							// Ask operator to fill calbox
							GVL_HMI.bCalBoxNeedsAttention := TRUE;
							bCalBoxAttention := TRUE;
	
							// Stop requesting until operator continues
							bRequestWeight := FALSE;
	
							eStepResume := E_CalibStep.CHECKING_WEIGH;
							eStep       := E_CalibStep.CALBOX_ATTENTION;
	
						ELSE
							// Proceed
							bBoxWeightOK := FALSE;
							bRequestWeight := FALSE;
	
							eStep := E_CalibStep.FEED_HMI_RESULTS;
							rAcceptanceCrit := GVL_Settings.stCalibParameters.rAcceptanceCriteria;
						END_IF
					END_IF
	
					// ------------------------------------------------
					// 4) Always reset the device session AFTER processing
					//    (so bWeightReady doesn't stay stuck TRUE / repeat)
					// ------------------------------------------------
					// If Reset() returns BOOL and you need to ensure completion, you can loop it outside.
					// For now, keep your pattern:
					GVL_Calibration.fbScaleDevice.Reset();
				END_IF
			END_IF
		END_IF
	
	E_CalibStep.FEED_HMI_RESULTS:
	
		FOR i := 1 TO 10 DO
			IF aPumpSettings[i].bSelected THEN
				GVL_HMI.aCalPumpResults[i].eStatus := E_CalibrationStatus.PENDING;
			END_IF
		END_FOR
		
		eStep := E_CalibStep.POSITION_MOTORS;
		
		
	E_CalibStep.POSITION_MOTORS:
	
		sStatus := 'Positioning motors M2 and M3';
		
		// Positioning motors M2 and M3 to calibration position 
		IF NOT bMoveMotorM3 THEN
			bMoveMotorM3 := GVL_Motion.aMotors[3].MoveAbsolute(GVL_Settings.stMachineParam.aM3Position[4], GVL_Settings.stMachineParam.rM3Velocity, GVL_Settings.stMachineParam.rM3Accleration, GVL_Settings.stMachineParam.rM3Deceleration);
		END_IF
		IF NOT bMoveMotorM2 AND bMoveMotorM3 THEN
			bMoveMotorM2 := GVL_Motion.aMotors[2].MoveAbsolute(GVL_Settings.stMachineParam.aM2Position[5], GVL_Settings.stMachineParam.rM2Velocity, GVL_Settings.stMachineParam.rM2Accleration, GVL_Settings.stMachineParam.rM2Deceleration);
		END_IF
	
		IF bMoveMotorM2 AND bMoveMotorM3 THEN
			tonMotorsDelay(in := TRUE, pt := T#200MS);
		END_IF
		
		IF tonMotorsDelay.Q THEN
			tonStepTimeout(IN := FALSE);
			eStep := E_CalibStep.POSITION_VALVES;
		END_IF

    E_CalibStep.POSITION_VALVES:
		//Reset Motors Flags
		bMoveMotorM2 := FALSE;
		bMoveMotorM3 := FALSE;	
		tonMotorsDelay(in := FALSE);
	
		tonStepTimeout(IN := TRUE, PT := tStepTimeout);
        sStatus := 'Positioning valves to Position 6';
		// Positioning the valves to the needles, position 6 
        FOR i := 1 TO 5 DO
            IF NOT bMoveValve[i] THEN
                bMoveValve[i] := GVL_Motion.aValvesObj[i].MoveValve(iPosition := 6, rVelocity := GVL_Motion.aValves[i].rTargetVel, rAcc := GVL_Motion.aValves[i].rAcceleration, rDec := GVL_Motion.aValves[i].rDeceleration);
            END_IF
        END_FOR
       IF bMoveValve[1] AND bMoveValve[2] AND bMoveValve[3] AND bMoveValve[4] AND bMoveValve[5] THEN
			FOR i := 1 TO 5 DO bMoveValve[i] := FALSE; END_FOR
			tonStepTimeout(IN := FALSE);
			eStep := E_CalibStep.FILLJAR_FORWARD; 
		ELSIF tonStepTimeout.Q THEN
			sStatus := 'Timeout while positioning valves';
			eStep := E_CalibStep.ERROR;
		END_IF

	E_CalibStep.FILLJAR_FORWARD:
		
		
		sStatus := CONCAT('Filling up the jar: ', F_JarName(iPumpIndex := iPumpIndex));
		
		IF aPumpSettings[iPumpIndex].bSelected THEN
			IF iPumpIndex = 1 THEN
				rFillJarTotalVol := aPumpSettings[iPumpIndex].rTargetVolume + GVL_Settings.stPumpParameters.iFillolventTubesFactor;
			ELSE
				rFillJarTotalVol := GVL_Settings.stPumpParameters.iFillolventTubesFactor;
			END_IF
			
			GVL_HMI.aCalPumpResults[iPumpIndex].eStatus := E_CalibrationStatus.RUNNING;
			
			//Move Motor M2 for IntoResBottom
			IF NOT bMoveMotorM2 THEN
				bMoveMotorM2 := GVL_Motion.aMotors[2].MoveAbsolute(GVL_Settings.stMachineParam.aM2Position[4], GVL_Settings.stMachineParam.rM2Velocity, GVL_Settings.stMachineParam.rM2Accleration, GVL_Settings.stMachineParam.rM2Deceleration);
			END_IF
				
			rDistanceByVol := F_VolumeToSteps_Path(rVolume := rFillJarTotalVol, iPumpIndex := iPumpIndex, ePath := E_PumpPath.FromCalBox);
			// Filling up the jar to start the calibration
			IF bMoveMotorM2 AND NOT bMovePump THEN
				bMovePump := GVL_Motion.aPumpsRotary[iPumpIndex].MoveRelative(	Distance := rDistanceByVol, 
																				Velocity := GVL_Settings.stPumpParameters.iMeterVelocity * 6, 	//RPM to Degree/sec
																				Acc := GVL_Settings.stPumpParameters.iMeterVelocity * 6,   		//RPM to Degree/sec
																				Dec := GVL_Settings.stPumpParameters.iMeterVelocity * 6			//RPM to Degree/sec
																			 );
			END_IF
	
			IF bMovePump THEN
				tonWeigthStabilization(IN := TRUE, PT := tWeightStable);
				sStatus := 'Waiting for weight stabilization...';
				IF tonWeigthStabilization.Q THEN
					bMovePump := FALSE;
					bMoveMotorM2 := FALSE;
					tonWeigthStabilization(IN := FALSE);
					bRequestWeight := TRUE;
					bWeightReady := FALSE;
					eStep := E_CalibStep.WEIGH_BEFORE;
				END_IF
			END_IF
		ELSE
			// If the pumps was not selected go to next one
			eStep := E_CalibStep.NEXT_PUMP;
		END_IF

	
    E_CalibStep.WEIGH_BEFORE:
		
        sStatus := CONCAT('Pump ', CONCAT(TO_STRING(iPumpIndex), CONCAT(' | Check ', CONCAT(TO_STRING(iReplicate + 1), ' | Taring Scale..'))));
		
		//Move Motor M2 for IntoResWEight
		IF NOT bMoveMotorM2 THEN
			bMoveMotorM2 := GVL_Motion.aMotors[2].MoveAbsolute(GVL_Settings.stMachineParam.aM2Position[6], GVL_Settings.stMachineParam.rM2Velocity, GVL_Settings.stMachineParam.rM2Accleration, GVL_Settings.stMachineParam.rM2Deceleration);
		END_IF
		
        IF bMoveMotorM2 AND bRequestWeight AND NOT bWeightReady THEN
            rScaleWeight := GVL_Calibration.fbScaleDevice.RequestWeight();
            IF GVL_Calibration.fbScaleDevice.bWeightReady THEN
                IF rScaleWeight = 9999.0 THEN
					tonCalDelay(IN := FALSE);
					tonStepTimeout(IN := FALSE);
					tonWeigthStabilization(IN := FALSE);
	
					GVL_HMI.bScaleNeedsAtention := TRUE;
					bScaleAttention := TRUE;
	
					bRequestWeight := FALSE;
					bWeightReady   := FALSE;
	
					eStepResume := E_CalibStep.WEIGH_BEFORE;
					eStep := E_CalibStep.SCALE_ATTENTION;
				ELSE
					rWeightBefore := rScaleWeight;
					
					GVL_calibration.stPumpCalibrationData[GVL_Calibration.iResultIndex].rTareWeigth := rWeightBefore;
					GVL_Calibration.stPumpCalibrationData[GVL_Calibration.iResultIndex].iPumpNumber := TO_USINT(iPumpIndex);
	
					bWeightReady   := TRUE;
					bRequestWeight := NOT GVL_Calibration.fbScaleDevice.Reset();
				END_IF
            END_IF
		END_IF
		IF bWeightReady THEN
			IF (rWeightBefore >= 0 AND rWeightBefore <= 1300) THEN
				GVL_calibration.stPumpCalibrationData[GVL_Calibration.iResultIndex].rTareWeigth := rWeightBefore;
				GVL_Calibration.stPumpCalibrationData[GVL_Calibration.iResultIndex].iPumpNumber := TO_USINT(iPumpIndex);
				rDistanceByVol := 0.0;
				bWeightReady := FALSE;
				bMoveMotorM2 := FALSE;
				eStep := E_CalibStep.WITHDRAW_BACKWARDS;
			ELSE
				eStep := E_CalibStep.ERROR;
			END_IF
		END_IF        

	
    E_CalibStep.WITHDRAW_BACKWARDS:

		sStatus := CONCAT(CONCAT('Pump ',CONCAT(TO_STRING(iPumpIndex),CONCAT(' | Check ',TO_STRING(iReplicate + 1)))),CONCAT(' | Pumping to calibration box: ',CONCAT(TO_STRING(aVolumeSetpoint[iPumpIndex]),' ml')));
		
		//Move Motor M2 for IntoResDispense
		IF NOT bMoveMotorM2 THEN
			bMoveMotorM2 := GVL_Motion.aMotors[2].MoveAbsolute(GVL_Settings.stMachineParam.aM2Position[5], GVL_Settings.stMachineParam.rM2Velocity, GVL_Settings.stMachineParam.rM2Accleration, GVL_Settings.stMachineParam.rM2Deceleration);
		END_IF
		
		aVolumeSetpoint[iPumpIndex] := aPumpSettings[iPumpIndex].rTargetVolume;

		GVL_calibration.stPumpCalibrationData[GVL_Calibration.iResultIndex].rTargetVolume := aPumpSettings[iPumpIndex].rTargetVolume;
		
		rDistanceByVol := F_VolumeToSteps_Path(rVolume := aVolumeSetpoint[iPumpIndex], iPumpIndex := iPumpIndex, ePath := E_PumpPath.FillCalBox );
		
		GVL_calibration.stPumpCalibrationData[GVL_Calibration.iResultIndex].iPumpRevs := TO_UINT(rDistanceByVol/360);
		GVL_HMI.aCalPumpResults[iPumpIndex].iRevsDone := GVL_calibration.stPumpCalibrationData[GVL_Calibration.iResultIndex].iPumpRevs; // Mirror pump revs done to the results table on HMI
		
		IF bMoveMotorM2 AND NOT bMovePump THEN
			bMovePump := GVL_Motion.aPumpsRotary[iPumpIndex].MoveRelative( 	Distance := - rDistanceByVol, 
																			Velocity := GVL_Settings.stPumpParameters.iMeterVelocity * 6, 	//RPM to Degree/sec
																			Acc := GVL_Settings.stPumpParameters.iMeterVelocity * 6, 		//RPM to Degree/sec
																			Dec := GVL_Settings.stPumpParameters.iMeterVelocity				//RPM to Degree/sec
																		 	);
		END_IF
		
		IF bMovePump THEN
			tonWeigthStabilization(in := TRUE, pt := tWeightStable);
			sStatus :='Waiting for weight stabilization...';
			IF bMoveMotorM2 AND tonWeigthStabilization.Q THEN
				bRequestWeight := TRUE;
				bMovePump := FALSE;
				bMoveMotorM2 := FALSE;
				tonWeigthStabilization(IN := FALSE);
				fbLocalSystemTime(bEnable := FALSE);
				bDTReady := FALSE;
				eStep := E_CalibStep.WEIGH_AFTER;
			END_IF
		END_IF


	
    E_CalibStep.WEIGH_AFTER:

		sStatus := CONCAT('Pump ', CONCAT(TO_STRING(iPumpIndex), CONCAT(' | Check ', CONCAT(TO_STRING(iReplicate + 1), ' | Requesting Gross Weight...'))));
	
		//Move Motor M2 for IntoResWeight
		IF NOT bMoveMotorM2 THEN
			bMoveMotorM2 := GVL_Motion.aMotors[2].MoveAbsolute(GVL_Settings.stMachineParam.aM2Position[6], GVL_Settings.stMachineParam.rM2Velocity, GVL_Settings.stMachineParam.rM2Accleration, GVL_Settings.stMachineParam.RM2Deceleration);
		END_IF
		
        IF bMoveMotorM2 AND bRequestWeight AND NOT bWeightReady THEN
            rScaleWeight := GVL_Calibration.fbScaleDevice.RequestWeight();
            IF GVL_Calibration.fbScaleDevice.bWeightReady THEN
                IF rScaleWeight = 9999.0 THEN
					tonCalDelay(IN := FALSE);
					tonStepTimeout(IN := FALSE);
					tonWeigthStabilization(IN := FALSE);
	
					GVL_HMI.bScaleNeedsAtention := TRUE;
					bScaleAttention := TRUE;
	
					bRequestWeight := FALSE;
					bWeightReady   := FALSE;
	
					eStepResume := E_CalibStep.WEIGH_AFTER;
					eStep := E_CalibStep.SCALE_ATTENTION;
				ELSE
					rWeightAfter := rScaleWeight;
					bWeightReady := TRUE;
					// NET (weight delta)
					rWeightDelta := rWeightAfter - rWeightBefore;
	
					// Mirror to logs
					GVL_calibration.stPumpCalibrationData[GVL_Calibration.iResultIndex].rGrossWeigth := rWeightAfter;
					GVL_calibration.stPumpCalibrationData[GVL_Calibration.iResultIndex].rNetWeigth := rWeightDelta;
	
					// Density-based volume
					GVL_calibration.stPumpCalibrationData[GVL_Calibration.iResultIndex].rNetVolume := rWeightDelta / rSolventDensity;
					
					rVolume := GVL_calibration.stPumpCalibrationData[GVL_Calibration.iResultIndex].rNetVolume;
					
					//Getting Sum Values to calculate the average on the end of replicates
					rPumpVolumeSum  := rPumpVolumeSum + rVolume;
					rTareWeightSum  := rTareWeightSum + rWeightBefore;
					rGrossWeightSum := rGrossWeightSum + rWeightAfter;
	
					bRequestWeight := NOT GVL_Calibration.fbScaleDevice.Reset();
				END_IF
			END_IF	
		END_IF	
		
		 // Produce a timestamp: DD-MMM-YYYY HH:MM:SS
        fbLocalSystemTime(bEnable := TRUE, dwCycle := 5);
		
        IF fbLocalSystemTime.bValid THEN
            stLocal := fbLocalSystemTime.systemTime;

            sMMo := F_MonthString(stLocal.wMonth);
            sDD  := F_TwoDigits(stLocal.wDay);
            sHH  := F_TwoDigits(stLocal.wHour);
            sMM  := F_TwoDigits(stLocal.wMinute);
            sSS  := F_TwoDigits(stLocal.wSecond);

			sStamp := CONCAT(sDD, '-');			//DD-
			sStamp := CONCAT(sStamp, sMMo);		//DD-MMM
			sStamp := CONCAT(sStamp, '-');		//DD-MMM-
			sStamp := CONCAT(sStamp, INT_TO_STRING(stLocal.wYear)); //DD-MMM-YYYY
			sStamp := CONCAT(sStamp, ' '); 		//DD-MMM-YYYY 
			sStamp := CONCAT(sStamp, sHH);		//DD-MMM-YYYY HH
			sStamp := CONCAT(sStamp, ':');		//DD-MMM-YYYY HH:
			sStamp := CONCAT(sStamp, sMM);		//DD-MMM-YYYY HH:MM
			sStamp := CONCAT(sStamp, ':');		//DD-MMM-YYYY HH:MM:
			sStamp := CONCAT(sStamp, sSS); 		//DD-MMM-YYYY HH:MM:SS

			bDTReady := TRUE;			
        ELSE
            sStamp := '00000000_000000'; // Fallback if system time is not valid
        END_IF
		
		IF bWeightReady AND bDTReady THEN
			
			rPercentDifference := ((rVolume - aPumpSettings[iPumpIndex].rTargetVolume)  / aPumpSettings[iPumpIndex].rTargetVolume) * 100;
			GVL_Calibration.stPumpCalibrationData[GVL_Calibration.iResultIndex].rDifferenceUl := rVolume - aPumpSettings[iPumpIndex].rTargetVolume;
			GVL_Calibration.stPumpCalibrationData[GVL_Calibration.iResultIndex].dDateTime := sStamp;
			GVL_Calibration.stPumpCalibrationData[GVL_Calibration.iResultIndex].rDifferencePercent := rPercentDifference;
			GVL_Calibration.stPumpCalibrationData[GVL_Calibration.iResultIndex].rCriteria := rAcceptanceCrit;
			
			//pupulate gross weight and net weight
			IF ABS(rPercentDifference) <= rAcceptanceCrit THEN
				aPumpResults[iPumpIndex].eStatus := E_CalibrationStatus.PASSED;
			ELSE
				// Adjust Needed flag 
				bPumpAdjustNeed := TRUE;
			END_IF
			
			iReplicate := iReplicate + 1;
			
			GVL_Calibration.stPumpCalibrationData[GVL_Calibration.iResultIndex].sStep := CONCAT('Check ', TO_STRING(iReplicate));
			
			//DB_Query.state:= E_DB_QUERY_STATE.INSERT_CALIBRATION_VALUES; //Insert new register of data on DB.
			GVL_Calibration.iResultIndex := GVL_Calibration.iResultIndex + 1;
			
			IF iReplicate >= GVL_Settings.stCalibParameters.iReplicatesSetpoint THEN
				
				// Calculating the average pump results
				rPumpAverageVolume  := rPumpVolumeSum / iReplicate;
				rPumpAvgTareWeigth  := rTareWeightSum / iReplicate;
				rPumpAvgGrossWeigth := rGrossWeightSum / iReplicate;
				
				// Mirror the pump status to HMI
				GVL_HMI.aCalPumpResults[iPumpIndex].rAvgNetVolume := rPumpAverageVolume;
				GVL_HMI.aCalPumpResults[iPumpIndex].rAvgTareWeight := rPumpAvgTareWeigth;
				GVL_HMI.aCalPumpResults[iPumpIndex].rAvgGrossWeight := rPumpAvgGrossWeigth;
				
				IF bPumpAdjustNeed THEN
					
					IF GVL_Calibration.iAllowableFailures > iNumberOfAdjusts THEN
						iReplicate := 0;
						iNumberOfAdjusts := iNumberOfAdjusts + 1;
						bPumpAdjustNeed := FALSE;
						DB_Query.state:= E_DB_QUERY_STATE.INSERT_CALIBRATION_VALUES; //Insert new register of data on DB.
						eStep := E_CalibStep.PUMPFACTOR_ADJUST;
					ELSE
						bPumpAdjustNeed := FALSE;
						eStep := E_CalibStep.PUMPFACTOR_FAILED;
					END_IF
					
				ELSE
					GVL_HMI.aCalPumpResults[iPumpIndex].eStatus := E_CalibrationStatus.PASSED;
					eStep := E_CalibStep.EMPTYJAR_BACKWARDS;
				END_IF
			ELSE
				eStep := E_CalibStep.RETURN_FORWARD;
			END_IF
			bMoveMotorM2 := FALSE;
			bWeightReady := FALSE;
		END_IF
		
	E_CalibStep.PUMPFACTOR_ADJUST: // Calculate the new factor
	
		IF NOT DB_Query.FB_Insert.bBusy AND bDataBaseSeq THEN
			GVL_Calibration.iResultIndex := GVL_Calibration.iResultIndex + 1;
			eStep := E_CalibStep.RETURN_FORWARD;
			bDataBaseSeq := FALSE;
		
		ELSIF NOT DB_Query.FB_Insert.bBusy AND NOT bDataBaseSeq THEN
			
			// Mirror the pump status to HMI
			GVL_HMI.aCalPumpResults[iPumpIndex].eStatus := E_CalibrationStatus.ADJUSTMENT_NEEDED;
			GVL_HMI.aCalPumpResults[iPumpIndex].rAvgNetVolume := rPumpAverageVolume;
			GVL_HMI.aCalPumpResults[iPumpIndex].rAvgTareWeight := rPumpAvgTareWeigth;
			GVL_HMI.aCalPumpResults[iPumpIndex].rAvgGrossWeight := rPumpAvgGrossWeigth;
			
			// new factor := target / Trunc((target / (Average / revs) ) + 0.5)  
			GVL_Retain.aCalibrationPumpFactor[iPumpindex] := aPumpSettings[iPumpIndex].rTargetVolume / TO_LREAL(TRUNC((aPumpSettings[iPumpIndex].rTargetVolume/(rPumpAverageVolume/GVL_calibration.stPumpCalibrationData[GVL_Calibration.iResultIndex - 1].iPumpRevs))+ 0.5));
			
			GVL_Motion.aPumps[iPumpindex].Rotary.rPumpFactorFillCalBox := GVL_Retain.aCalibrationPumpFactor[iPumpindex];
			GVL_Motion.aPumps[iPumpindex].Rotary.rPumpFactorFillJars   := GVL_Retain.aCalibrationPumpFactor[iPumpindex];
			GVL_Motion.aPumps[iPumpindex].Rotary.rPumpFactorFromCalBox := GVL_Retain.aCalibrationPumpFactor[iPumpindex];
			
			// Populate the adjustment row	
			GVL_Calibration.stPumpCalibrationData[GVL_Calibration.iResultIndex].iPumpNumber := TO_USINT(iPumpIndex);
			GVL_Calibration.stPumpCalibrationData[GVL_Calibration.iResultIndex].sStep := 'Adjustment';
			GVL_Calibration.stPumpCalibrationData[GVL_Calibration.iResultIndex].dDateTime := sStamp;
			GVL_Calibration.stPumpCalibrationData[GVL_Calibration.iResultIndex].rTareWeigth := 0.00;
	
			GVL_calibration.stPumpCalibrationData[GVL_Calibration.iResultIndex].rGrossWeigth := 0.00;
	
			GVL_calibration.stPumpCalibrationData[GVL_Calibration.iResultIndex].rNetWeigth := 0.00;
			
	
			GVL_Calibration.stPumpCalibrationData[GVL_Calibration.iResultIndex].rNetVolume := 0.00;
	
			GVL_Calibration.stPumpCalibrationData[GVL_Calibration.iResultIndex].rTargetVolume := 0.00;
			GVL_Calibration.stPumpCalibrationData[GVL_Calibration.iResultIndex].rDifferencePercent := 0.00;
			
			GVL_Calibration.stPumpCalibrationData[GVL_Calibration.iResultIndex].rCriteria := 0.00;
			GVL_Calibration.stPumpCalibrationData[GVL_Calibration.iResultIndex].iPumpRevs := TO_UINT(aPumpSettings[iPumpIndex].rTargetVolume / GVL_Motion.aPumps[iPumpindex].Rotary.rPumpFactorFillCalBox);	
			
			// final transition
			rPumpAverageVolume := 0.00;
			rPumpAvgTareWeigth := 0.00;
			rPumpAvgGrossWeigth := 0.00;
			rPumpVolumeSum := 0.00;
			rTareWeightSum := 0.00;
			rGrossWeightSum := 0.00;
			iReplicate := 0;
			
			DB_Query.state:= E_DB_QUERY_STATE.INSERT_CALIBRATION_VALUES; //Insert new register of data on DB.
			bDataBaseSeq := TRUE;
		END_IF
		
		
	E_CalibStep.PUMPFACTOR_FAILED:
		// Update the HMI pump status
		GVL_HMI.aCalPumpResults[iPumpIndex].eStatus := E_CalibrationStatus.FAILED;
		GVL_HMI.aCalPumpResults[iPumpIndex].rAvgNetVolume := rPumpAverageVolume;
		GVL_HMI.aCalPumpResults[iPumpIndex].rAvgTareWeight := rPumpAvgTareWeigth;
		GVL_HMI.aCalPumpResults[iPumpIndex].rAvgGrossWeight := rPumpAvgGrossWeigth;
		
		// Changing the Step string to have failed in it
		GVL_Calibration.stPumpCalibrationData[GVL_Calibration.iResultIndex - 1].sStep := CONCAT(CONCAT('Check ', TO_STRING(iReplicate)), CONCAT(' ***', CONCAT(CHR(13) , CONCAT(CHR(10), 'FAILED ***'))));
		
		// final transition
		iNumberOfAdjusts := 0;
		rPumpAverageVolume := 0.00;
		rPumpAvgTareWeigth := 0.00;
		rPumpAvgGrossWeigth := 0.00;
		rPumpVolumeSum := 0.00;
		rTareWeightSum := 0.00;
		rGrossWeightSum := 0.00;
		iReplicate := 0;
		eStep := E_CalibStep.EMPTYJAR_BACKWARDS;
		
    E_CalibStep.RETURN_FORWARD:

		sStatus := CONCAT(CONCAT('Pump ',CONCAT(TO_STRING(iPumpIndex), CONCAT(' | Check ', CONCAT(TO_STRING(iReplicate + 1), ' | ')))), CONCAT('Returning solvent back to the Jar : ', F_JarName(iPumpIndex := iPumpIndex)));
		rDistanceByVol := F_VolumeToSteps_Path(rVolume := (aPumpSettings[iPumpIndex].rTargetVolume + 5), iPumpIndex := iPumpIndex, ePath := E_PumpPath.FromCalBox);
		
		//Move Motor M2 for IntoResWeight
		IF NOT bMoveMotorM2 THEN
			bMoveMotorM2 := GVL_Motion.aMotors[2].MoveAbsolute(GVL_Settings.stMachineParam.aM2Position[4], GVL_Settings.stMachineParam.rM2Velocity, GVL_Settings.stMachineParam.rM2Accleration, GVL_Settings.stMachineParam.rM2Deceleration);
		END_IF
			
        IF bMoveMotorM2 AND NOT bMovePump THEN
			bMovePump := GVL_Motion.aPumpsRotary[iPumpIndex].MoveRelative( 	Distance := rDistanceByVol, 
																			Velocity := GVL_Settings.stPumpParameters.iMeterVelocity * 6, 	//RPM to Degree/sec
																			Acc := GVL_Settings.stPumpParameters.iMeterVelocity * 6, 		//RPM to Degree/sec
																			Dec := GVL_Settings.stPumpParameters.iMeterVelocity * 6			//RPM to Degree/sec
																		  	);
		END_IF
		
		IF bMovePump THEN
			tonWeigthStabilization(IN := TRUE, PT := tWeightStable);
			sStatus := 'Waiting for weight stabilization...';
			IF tonWeigthStabilization.Q THEN
				bMovePump := FALSE;
				bMoveMotorM2 := FALSE;
				tonWeigthStabilization(IN := FALSE);
				bRequestWeight := TRUE;
				bWeightReady := FALSE;
				eStep := E_CalibStep.WEIGH_BEFORE; // Starts next replication
			END_IF
		END_IF
		DB_Query.state:= E_DB_QUERY_STATE.INSERT_CALIBRATION_VALUES; //Insert new register of data on DB.
		
	E_CalibStep.EMPTYJAR_BACKWARDS:

		sStatus := CONCAT('Pump ',CONCAT(TO_STRING(iPumpIndex),CONCAT(' | Empty the jar number: ',TO_STRING(iPumpIndex))));
		aVolumeSetpoint[iPumpIndex] := aPumpSettings[iPumpIndex].rTargetVolume;
		
		//Move Motor M2 for IntoResDispense
		IF NOT bMoveMotorM2 THEN
			bMoveMotorM2 := GVL_Motion.aMotors[2].MoveAbsolute(GVL_Settings.stMachineParam.aM2Position[5], GVL_Settings.stMachineParam.rM2Velocity, GVL_Settings.stMachineParam.rM2Accleration, GVL_Settings.stMachineParam.rM2Deceleration);
		END_IF
		(*
		IF iPumpIndex = 1 THEN
			rEmptyJarTotalVol := aVolumeSetpoint[iPumpIndex] + GVL_Settings.stPumpParameters.iEmptyFactor;
		ELSE
			rEmptyJarTotalVol := GVL_Settings.stPumpParameters.iEmptyFactor;
		END_IF
		*)
		
		rEmptyJarTotalVol := aVolumeSetpoint[iPumpIndex] + GVL_Settings.stPumpParameters.iEmptyFactor;
		
		rDistanceByVol := F_VolumeToSteps_Path(rVolume := rEmptyJarTotalVol, iPumpIndex := iPumpIndex, ePath := E_PumpPath.FromCalBox );
		
        IF bMoveMotorM2 AND NOT bMovePump THEN
			bMovePump := GVL_Motion.aPumpsRotary[iPumpIndex].MoveRelative( 	Distance := - rDistanceByVol, 
																			Velocity := GVL_Settings.stPumpParameters.iRunVelocity * 6, 	//RPM to Degree/sec
																			Acc := GVL_Settings.stPumpParameters.iRunVelocity * 6, 			//RPM to Degree/sec
																			Dec := GVL_Settings.stPumpParameters.iRunVelocity * 6			//RPM to Degree/sec
																		  	);
		END_IF
		
		IF bMovePump THEN
			bMoveMotorM2 := FALSE;
			bMovePump := FALSE;
			eStep := E_CalibStep.NEXT_PUMP;
		END_IF
		DB_Query.state:= E_DB_QUERY_STATE.INSERT_CALIBRATION_VALUES; //Insert new register of data on DB.
	
    E_CalibStep.NEXT_PUMP:
		// Reset sum and avg values	
        iPumpIndex := iPumpIndex + 1;
        iReplicate := 0;
		iNumberOfAdjusts := 0;
		rPumpAverageVolume := 0.00;
		rPumpAvgTareWeigth := 0.00;
		rPumpAvgGrossWeigth := 0.00;
		rPumpVolumeSum := 0.00;
		rTareWeightSum := 0.00;
		rGrossWeightSum := 0.00;
        IF iPumpIndex <= 10 THEN
            eStep := E_CalibStep.FILLJAR_FORWARD;
        ELSE
            eStep := E_CalibStep.HOMING_MOTORS;
        END_IF

	
    E_CalibStep.HOMING_MOTORS:
        sStatus := 'Returning M2 and M3 to home';
				
		IF NOT bMoveMotorM2 THEN
			bMoveMotorM2 := GVL_Motion.aMotors[2].MoveAbsolute(	GVL_Settings.stMachineParam.aM2Position[1], 
																GVL_Settings.stMachineParam.rM2Velocity, 
																GVL_Settings.stMachineParam.rM2Accleration, 
																GVL_Settings.stMachineParam.rM2Deceleration
																);
		END_IF
		IF NOT bMoveMotorM3 AND bMoveMotorM2 THEN
			bMoveMotorM3 := GVL_Motion.aMotors[3].MoveAbsolute(	GVL_Settings.stMachineParam.aM3Position[1], 
																GVL_Settings.stMachineParam.rM3Velocity, 
																GVL_Settings.stMachineParam.rM3Accleration, 
																GVL_Settings.stMachineParam.rM3Deceleration
																);
		END_IF
				
		IF bMoveMotorM2 AND bMoveMotorM3 THEN
			tonMotorsDelay(in := TRUE, pt := T#200MS);
		END_IF
		
		IF tonMotorsDelay.Q THEN
			tonStepTimeout(IN := FALSE);
			IF GVL_Settings.stCalibParameters.iAirDryTimeSec > 0 THEN // IF Air Dry time settings is greater than zero go to air dry step
				eStep := E_CalibStep.REPORT_INFO_UPDATE; // AIR_DRY_TIME
			ELSE
				eStep := E_CalibStep.REPORT_INFO_UPDATE;
			END_IF
		END_IF
   
		
	E_CalibStep.AIR_DRY_TIME:
		IF NOT bSetSolenoids THEN
			//Check if the M1 motor is not on seal stages position
			IF GVL_Settings.stMachineParam.aM1Position[2] >= (GVL_Motion.M1Motor.rActualPos + rPosTolerance) AND NOT bMoveMotorM1 THEN
				IF NOT bMoveMotorM1 THEN
					bMoveMotorM1 := NOT GVL_Motion.aMotors[1].MoveAbsolute(	rPosition := GVL_Settings.stMachineParam.aM1Position[2],
																			rVelocity := GVL_Settings.stMachineParam.rM1Velocity,
																			rAcc	  := GVL_Settings.stMachineParam.rM1Accleration,
																			rDec	  := GVL_Settings.stMachineParam.rM1Deceleration);
				END_IF
			ELSE
				//M1 Position ok
				bSetSolenoids := GVL_IO.gSetSolenoidControl.AirDry(); //Open Solenoids
				bMoveMotorM1 := TRUE;
			END_IF
		ELSE
			bMoveMotorM1 := FALSE;
			bAirDryTrigger := TRUE;
		END_IF
		
		// Air Dry Timer
		tonAirDry( IN := bAirDryTrigger, PT := UINT_TO_TIME(GVL_Settings.stCalibParameters.iAirDryTimeSec*1000));
		
		IF tonAirDry.Q THEN
			//Return Solenoids to Idle state
			IF GVL_IO.gSetSolenoidControl.Idle() THEN
				bSetSolenoids := FALSE;
				//Transition
				eStep := E_CalibStep.REPORT_INFO_UPDATE;
			END_IF
		END_IF
	
	E_CalibStep.REPORT_INFO_UPDATE: //TODO: Update the variables without hardcode
		//Reset Motors Flags
		bMoveMotorM2 := FALSE;
		bMoveMotorM3 := FALSE;	
		tonMotorsDelay(in := FALSE);
		
		//Report Info
		GVL_Calibration.stPumpCalReportInfo.sReportName := GVL_Constant.sPumpCalibrationReportName;
		GVL_Calibration.stPumpCalReportInfo.sReoportSubName := GVL_Constant.sPumpCalibrationReportSubName;
		GVL_Calibration.stPumpCalReportInfo.sDatabaseName := GVL_Constant.sDatabaseName;
		GVL_Calibration.stPumpCalReportInfo.sReportDate := sStamp;
		GVL_Calibration.stPumpCalReportInfo.sPrintedBy := 'Administrator';
		GVL_Calibration.stPumpCalReportInfo.sSystemID := GVL_Constant.sSystemID;
		GVL_Calibration.stPumpCalReportInfo.iPage := 0;
		
		//Calibration Info
		GVL_Retain.iCalibrationNumber := GVL_Retain.iCalibrationNumber + 1;
		//GVL_Calibration.stPumpCalibrationInfo.iCalibrationNumber := TO_UINT(GVL_Retain.iCalibrationNumber);
		GVL_Calibration.stPumpCalibrationInfo.iAllowableFailures := GVL_Calibration.iAllowableFailures;
		GVL_Calibration.stPumpCalibrationInfo.iCalIntervalDays := 0;
		GVL_Calibration.stPumpCalibrationInfo.iReplicates := GVL_Calibration.iReplicatesSetpoint;
		GVL_Calibration.stPumpCalibrationInfo.iSolventID := GVL_Settings.stSolventsInfo[iSolvent].sSolventName;
		GVL_Calibration.stPumpCalibrationInfo.iSysMasterListRev := 0;
		GVL_Calibration.stPumpCalibrationInfo.iSysSettingsRev := 0;
		GVL_Calibration.stPumpCalibrationInfo.iUserID := 'vd24';
		
		eStep := E_CalibStep.COMPLETE; 		
		
	E_CalibStep.CALBOX_ATTENTION:
    // Pause here while the operator adjusts the box weight on the scale.
    // No timeouts are running in this state.

    bBusy   := TRUE;
    sStatus := 'Calibration box requires attention. Please fix and press continue.';

    // Continue pressed on HMI?
    IF GVL_HMI.bCalBoxFixed THEN
        // Clear HMI flags
        GVL_HMI.bCalBoxNeedsAttention := FALSE;
        GVL_HMI.bCalBoxFixed := FALSE;

        bCalBoxAttention := FALSE;

        // Re-arm the same step to re-request a fresh weight
        bRequestWeight := TRUE;
        bWeightReady   := FALSE;

        // Return exactly where we paused (CHECKING_WEIGH)
        eStep := eStepResume;

		ELSIF GVL_Calibration.bAbortCalibration THEN
			sStatus := 'Calibration aborted during calibration box attention.';
			eStep   := E_CalibStep.ERROR;
		END_IF	
		
	E_CalibStep.SCALE_ATTENTION:
		bBusy := TRUE;
		sStatus := 'Scale requires attention. Please fix on the device and press Continue.';
		
		// Resets calibration box attention
		GVL_HMI.bCalBoxNeedsAttention := FALSE;
		GVL_HMI.bCalBoxFixed := FALSE;
		bCalBoxAttention := FALSE;
		
		// Wait for operator to press "Continue" (HMI toggles this)
		IF GVL_HMI.bScaleFixed THEN
			GVL_HMI.bScaleNeedsAtention := FALSE;
			GVL_HMI.bScaleFixed := FALSE;
			bScaleAttention := FALSE;
	
			// Re-arm reading for the same step
			bRequestWeight := TRUE;
			bWeightReady   := FALSE;
	
			// Resume exactly where we were
			eStep := eStepResume;
	
		ELSIF GVL_Calibration.bAbortCalibration THEN
			sStatus := 'Calibration aborted during scale attention.';
			eStep := E_CalibStep.ERROR;
		END_IF
	
		
    E_CalibStep.COMPLETE:
        sStatus := 'Calibration Complete';
		iDataCount := GVL_Calibration.iResultIndex - 1;
        bDone := TRUE;
        bBusy := FALSE;
		
        // Remains here till external reset
	
    E_CalibStep.ERROR:
        bBusy := FALSE;
        bDone := FALSE;
        sStatus := 'Calibration aborted due to error. Press Stop button to start over';
		
		// FIX: The header row was already inserted into [CALIBRATION_HEAD] at
		// calibration start. If no measurements were recorded (iResultIndex <= 1),
		// that header row is now orphaned — it appears in the view with NULL
		// date columns because [CALIBRATION] has no matching rows.
		// Delete the orphaned header row so the view stays clean.
		IF iResultIndex <= 1 AND DB_Query.state = E_DB_QUERY_STATE.IDLE_STATE THEN
			DB_Query.state := E_DB_QUERY_STATE.DELETE_CALIBRATION_HEAD;
		END_IF
		
		// Remains here till external reset

END_CASE

ACT_ProgressUI_Real();

ACTION ACT_CleanStart:
iPumpIndex := 1;
iReplicate := 0;
iNumberOfAdjusts := 0;
GVL_Calibration.iResultIndex := 1; // first log row
rPumpAverageVolume := 0.00;
rPumpAvgTareWeigth := 0.00;
rPumpAvgGrossWeigth := 0.00;
rPumpVolumeSum := 0.00;
rTareWeightSum := 0.00;
rGrossWeightSum := 0.00;
bPumpAdjustNeed := FALSE;
bStartCalibration := FALSE;

FOR i := 1 TO 10 DO
	GVL_HMI.aCalPumpResults[i].eStatus := E_CalibrationStatus.IDLE;
	GVL_HMI.aCalPumpResults[i].rAvgNetVolume := 0.00;
	GVL_HMI.aCalPumpResults[i].rAvgTareWeight := 0.00;
	GVL_HMI.aCalPumpResults[i].rAvgGrossWeight := 0.00;
END_FOR
END_ACTION

ACTION ACT_ProgressUI_Real:
// --- 1) Detecta troca de sStatus e define PT com base real ---
IF sStatus <> sPrev THEN
    tPT := T#0MS; // default: sem barra
	
	// START DELAY
    IF (eStep = E_CalibStep.DELAY) OR (FIND(sStatus, 'Waiting delay') = 1) THEN
        tPT := tDelayStart;
	
    // POSITION_MOTORS  (usa |alvo - atual| / vel e pega o mais lento + 200ms)
    ELSIF FIND(sStatus, 'Positioning motors M2 and M3') = 1 THEN
        rDeltaM2 := ABS(GVL_Settings.stMachineParam.aM2Position[4] - GVL_Motion.M2Motor.rActualPos);
        rDeltaM3 := ABS(GVL_Settings.stMachineParam.aM3Position[4] - GVL_Motion.M3Motor.rActualPos); 
        rVM2 := MAX(0.1, GVL_Settings.stMachineParam.rM2Velocity);
        rVM3 := MAX(0.1, GVL_Settings.stMachineParam.rM3Velocity);
        rSecs := MAX(rDeltaM2 / rVM2, rDeltaM3 / rVM3) + 0.2;
        tPT := F_sec_to_time(rSecs);

    ELSIF FIND(sStatus, 'Positioning valves to Position 6') = 1 THEN
        tPT := T#2S;

    ELSIF FIND(sStatus, 'Filling up the jar') = 1 THEN
        rPumpVelDeg := MAX(1.0, GVL_Settings.stPumpParameters.iMeterVelocity) * 6.0; // RPM->deg/s
        rSecs := ABS(rDistanceByVol) / rPumpVelDeg;
        tPT := F_sec_to_time(rSecs);

    ELSIF (FIND(sStatus, 'Taring Scale') > 0) OR (FIND(sStatus, 'Requesting Gross Weight') = 1) THEN
        tPT := T#3S;

    ELSIF FIND(sStatus, 'Pumping to calibration box') > 0 THEN
        rPumpVelDeg := MAX(1.0, GVL_Settings.stPumpParameters.iMeterVelocity) * 6.0;
        rSecs := ABS(rDistanceByVol) / rPumpVelDeg;
        tPT := F_sec_to_time(rSecs);

    ELSIF FIND(sStatus, 'Returning solvent back to the Jar') > 0 THEN
        rPumpVelDeg := MAX(1.0, GVL_Settings.stPumpParameters.iMeterVelocity) * 6.0;
        rSecs := ABS(rDistanceByVol) / rPumpVelDeg;
        tPT := F_sec_to_time(rSecs);

    ELSIF FIND(sStatus, 'Empty the jar') = 1 THEN
        rRunVelDeg := MAX(1.0, GVL_Settings.stPumpParameters.iRunVelocity) * 6.0;
        rSecs := ABS(rDistanceByVol) / rRunVelDeg;
        tPT := F_sec_to_time(rSecs);

    ELSIF FIND(sStatus, 'Returning M2 and M3 to home') = 1 THEN
        rDeltaM2 := ABS(GVL_Settings.stMachineParam.aM2Position[1] - GVL_Motion.M2Motor.rActualPos);
        rDeltaM3 := ABS(GVL_Settings.stMachineParam.aM3Position[1] - GVL_Motion.M3Motor.rActualPos);
        rVM2 := MAX(0.1, GVL_Settings.stMachineParam.rM2Velocity);
        rVM3 := MAX(0.1, GVL_Settings.stMachineParam.rM3Velocity);
        rSecs := MAX(rDeltaM2 / rVM2, rDeltaM3 / rVM3) + 0.2;
        tPT := F_sec_to_time(rSecs);

    ELSIF (eStep = E_CalibStep.AIR_DRY_TIME) THEN
        tPT := UINT_TO_TIME(GVL_Settings.stCalibParameters.iAirDryTimeSec * 1000);

    ELSIF FIND(sStatus, 'Waiting for weight stabilization') = 1 THEN
        tPT := tonWeigthStabilization.PT;
    END_IF

    // Atualiza label na HMI
    GVL_HMI.sCalibProgressLabel := sStatus;

    // (Re)arma a barra
    IF tPT > T#0MS THEN
        GVL_HMI.bCalibStepLoading := TRUE;
        GVL_HMI.rCalibStepPercent := 0.0;

        // reset do TON (será armado novamente abaixo)
        tonProgress(IN := FALSE);
    ELSE
        GVL_HMI.bCalibStepLoading := FALSE;
        GVL_HMI.rCalibStepPercent := 0.0;
        tonProgress(IN := FALSE);
    END_IF
END_IF;

// --- 2) Chama SEMPRE o TON (enquanto loading estiver ativo) ---
tonProgress(
    IN := GVL_HMI.bCalibStepLoading,
    PT := tPT
);

// --- 3) Atualiza percentual enquanto carrega ---
IF GVL_HMI.bCalibStepLoading AND (tPT > T#0MS) THEN
    GVL_HMI.rCalibStepPercent :=
        LIMIT(0.0, 100.0 * TO_REAL(tonProgress.ET) / TO_REAL(tPT), 100.0);

    IF tonProgress.Q THEN
        GVL_HMI.rCalibStepPercent := 100.0;
        // GVL_HMI.bCalibStepLoading := FALSE;
        // tonProgress(IN := FALSE);
    END_IF
END_IF;

// --- 4) Memoriza último status ---
sPrev := sStatus;
END_ACTION

METHOD Reset : BOOL
VAR_INPUT
	bHard : BOOL := FALSE;
END_VAR
VAR
	iLocal : INT;
END_VAR
// 1) Stop motion/actuators best-effort (ignore returns; repeated calls are safe)
(*
IF (SIZEOF(GVL_Motion.aMotors) >= 3*SIZEOF(GVL_Motion.aMotors[1])) THEN
    GVL_Motion.aMotors[2].Stop();
    GVL_Motion.aMotors[3].Stop();
	GVL_Motion.aMotors[2].Reset();
	GVL_Motion.aMotors[3].Reset();
END_IF

FOR iLocal := 1 TO 10 DO
    GVL_Motion.aPumpsRotary[iLocal].Stop();
	GVL_Motion.aPumpsRotary[iLocal].Reset();
END_FOR

FOR iLocal := 1 TO 5 DO
    GVL_Motion.aValvesObj[iLocal].Stop();
	GVL_Motion.aValvesObj[iLocal].Reset();
END_FOR
*)

FOR iLocal := 1 TO 10 DO
	GVL_HMI.aCalPumpResults[iLocal].eStatus := E_CalibrationStatus.IDLE;
END_FOR

GVL_Calibration.fbScaleDevice.Reset();

// 2) Disarm timers/edge detectors and clear triggers
tonCalDelay(IN := FALSE);
tonStepTimeout(IN := FALSE);
tonWeigthStabilization(IN := FALSE);
tonMotorsDelay(in := FALSE);
tonProgress(in := FALSE);

// Drop R_TRIG by passing CLK := FALSE this cycle
bExecutePulse(CLK := FALSE);

// 3) Clear internal flags and intermediate states
bStartCalibration     := FALSE;
bCalibrationRequested := FALSE;

bRequestWeight        := FALSE;
bWeightReady          := FALSE;

bMovePump             := FALSE;
bMoveMotorM2          := FALSE;
bMoveMotorM3          := FALSE;
bDataBaseSeq 		  := FALSE;

FOR iLocal := 1 TO 5 DO
    bMoveValve[iLocal] := FALSE;
END_FOR

// 4) Reset indexes and temporaries
iPumpIndex    := 1;
iReplicate    := 0;
iResultIndex  := 1;
iNumberOfAdjusts := 0;

rWeightBefore 	 := 0.0;
rWeightAfter  	 := 0.0;
rWeightDelta  	 := 0.0;
rVolume       	 := 0.0;
rScaleWeight  	 := 0.0;
rDistanceByVol   := 0.0;
rFillJarTotalVol := 0.0;

rPumpAverageVolume := 0.00;
rPumpAvgTareWeigth := 0.00;
rPumpAvgGrossWeigth := 0.00;
rPumpVolumeSum := 0.00;
rTareWeightSum := 0.00;
rGrossWeightSum := 0.00;

sPrev       := '';
tPT         := T#0S;
rDeltaM2	:= 0.00;
rDeltaM3	:= 0.00;
rVM2		:= 0.00;
rVM3		:= 0.00;
rPumpVelDeg := 0.00;
rRunVelDeg	:= 0.00;
rSecs		:= 0.00;

// 5) Optional “hard” cleanup: clear selections and results
IF bHard THEN
    FOR iLocal := 1 TO 10 DO
        aPumpMask[iLocal]       := FALSE;
        aVolumeSetpoint[iLocal] := 0.0;
        aVelocity[iLocal]       := 0.0;
        aDirection[iLocal]      := E_PumpDirection.Forward; // default

        // Public result mirror (if you want a clean slate)
        aPumpResults[iLocal].eStatus        := E_CalibrationStatus.UNKNOWN;
        aPumpResults[iLocal].bAdjustment    := FALSE;
        aPumpResults[iLocal].bBusy          := FALSE;
        aPumpResults[iLocal].bSelected      := FALSE;
        aPumpResults[iLocal].iFailures      := 0;
        aPumpResults[iLocal].rActualVolume  := 0.0;
        aPumpResults[iLocal].rTargetVolume  := 0.0;
        aPumpResults[iLocal].tElapsed       := T#0S;
        aPumpResults[iLocal].tStartTime     := T#0S;

        // If you mirror HMI results elsewhere, clear here as needed.
    END_FOR
END_IF

// 6) Normalize outputs and step
bBusy   := FALSE;
bDone   := FALSE;
sStatus := 'Idle (reset)';
GVL_HMI.bAbortCalibrationBT := FALSE;
eStep   := E_CalibStep.IDLE;

// 7) Idempotent return
Reset := TRUE;
END_METHOD

END_FUNCTION_BLOCK

// ---- POUs/MotionControl/FB_AllPumpsController.TcPOU
FUNCTION_BLOCK FB_AllPumpsController
VAR_INPUT
END_VAR
VAR_OUTPUT
END_VAR
VAR
	bRequestMoveBySpeed		: BOOL := FALSE;
	bRequestMoveByVol		: BOOL := FALSE;
	bRequestMoveByDistance	: BOOL := FALSE;
	bRequestStopAllPumps	: BOOL := FALSE;
	bRequestMoveLinearPumps : BOOL := FALSE;
	
	bMoveVelocityPumps	: ARRAY[1..10] OF BOOL;
	bMoveDistancePumps	: ARRAY[1..10] OF BOOL;
	bMoveRelativePumps	: ARRAY[1..10] OF BOOL;
	bMoveLinearPumps	: ARRAY[1..10] OF BOOL;
	bStopRotaryPump 	: ARRAY[1..10] OF BOOL;
	bStopLinearPump		: ARRAY[1..10] OF BOOL;
	
	rDistanceByVol		: ARRAY[1..10] OF LREAL;
	aValvePosition		: ARRAY[1..10] OF SINT;
	aPumpPath			: ARRAY[1..10] OF E_PumpPath;
	
END_VAR

METHOD MoveByDistance : BOOL
VAR_INPUT
	aPumpIds		: ARRAY[1..10] OF BOOL;
	aPumpDirection 	: ARRAY[1..10] OF E_PumpDirection;
	aVelocity 		: ARRAY[1..10] OF REAL;
	aRevolutions	: ARRAY[1..10] OF UINT;
END_VAR
IF NOT bRequestMoveByDistance THEN
	MoveByDistance := FALSE;
	bMoveDistancePumps := aPumpIds;
	bRequestMoveByDistance := TRUE;
END_IF

//getting pump factor in mL/rev and converting to uL/degrees.
rDistanceByVol[1] := aRevolutions[1] * 360;
rDistanceByVol[2] := aRevolutions[2] * 360;
rDistanceByVol[3] := aRevolutions[3] * 360;
rDistanceByVol[4] := aRevolutions[4] * 360;
rDistanceByVol[5] := aRevolutions[5] * 360;
rDistanceByVol[6] := aRevolutions[6] * 360;
rDistanceByVol[7] := aRevolutions[7] * 360;
rDistanceByVol[8] := aRevolutions[8] * 360;
rDistanceByVol[9] := aRevolutions[9] * 360;
rDistanceByVol[10] := aRevolutions[10] * 360;

//Inverting the distance based on pumps flow direction
IF aPumpDirection[1] = E_PumpDirection.Backward THEN
	rDistanceByVol[1] := rDistanceByVol[1] * -1;
END_IF
IF aPumpDirection[2] = E_PumpDirection.Backward THEN
	rDistanceByVol[2] := rDistanceByVol[2] * -1;
END_IF
IF aPumpDirection[3] = E_PumpDirection.Backward THEN
	rDistanceByVol[3] := rDistanceByVol[3] * -1;
END_IF
IF aPumpDirection[4] = E_PumpDirection.Backward THEN
	rDistanceByVol[4] := rDistanceByVol[4] * -1;
END_IF
IF aPumpDirection[5] = E_PumpDirection.Backward THEN
	rDistanceByVol[5] := rDistanceByVol[5] * -1;
END_IF
IF aPumpDirection[6] = E_PumpDirection.Backward THEN
	rDistanceByVol[6] := rDistanceByVol[6] * -1;
END_IF
IF aPumpDirection[7] = E_PumpDirection.Backward THEN
	rDistanceByVol[7] := rDistanceByVol[7] * -1;
END_IF
IF aPumpDirection[8] = E_PumpDirection.Backward THEN
	rDistanceByVol[8] := rDistanceByVol[8] * -1;
END_IF
IF aPumpDirection[9] = E_PumpDirection.Backward THEN
	rDistanceByVol[9] := rDistanceByVol[9] * -1;
END_IF
IF aPumpDirection[10] = E_PumpDirection.Backward THEN
	rDistanceByVol[10] := rDistanceByVol[10] * -1;
END_IF

//Pumps relative movement
IF bMoveDistancePumps[1] THEN
	bMoveDistancePumps[1] := NOT GVL_Motion.aPumpsRotary[1].MoveRelative(Distance := rDistanceByVol[1], Velocity := aVelocity[1], Acc := aVelocity[1], Dec := aVelocity[1]);
END_IF
IF bMoveDistancePumps[2] THEN
	bMoveDistancePumps[2] := NOT GVL_Motion.aPumpsRotary[2].MoveRelative(Distance := rDistanceByVol[2], Velocity := aVelocity[2], Acc := aVelocity[2], Dec := aVelocity[2]);
END_IF
IF bMoveDistancePumps[3] THEN
	bMoveDistancePumps[3] := NOT GVL_Motion.aPumpsRotary[3].MoveRelative(Distance := rDistanceByVol[3], Velocity := aVelocity[3], Acc := aVelocity[3], Dec := aVelocity[3]);
END_IF
IF bMoveDistancePumps[4] THEN
	bMoveDistancePumps[4] := NOT GVL_Motion.aPumpsRotary[4].MoveRelative(Distance := rDistanceByVol[4], Velocity := aVelocity[4], Acc := aVelocity[4], Dec := aVelocity[4]);
END_IF
IF bMoveDistancePumps[5] THEN
	bMoveDistancePumps[5] := NOT GVL_Motion.aPumpsRotary[5].MoveRelative(Distance := rDistanceByVol[5], Velocity := aVelocity[5], Acc := aVelocity[5], Dec := aVelocity[5]);
END_IF
IF bMoveDistancePumps[6] THEN
	bMoveDistancePumps[6] := NOT GVL_Motion.aPumpsRotary[6].MoveRelative(Distance := rDistanceByVol[6], Velocity := aVelocity[6], Acc := aVelocity[6], Dec := aVelocity[6]);
END_IF
IF bMoveDistancePumps[7] THEN
	bMoveDistancePumps[7] := NOT GVL_Motion.aPumpsRotary[7].MoveRelative(Distance := rDistanceByVol[7], Velocity := aVelocity[7], Acc := aVelocity[7], Dec := aVelocity[7]);
END_IF
IF bMoveDistancePumps[8] THEN
	bMoveDistancePumps[8] := NOT GVL_Motion.aPumpsRotary[8].MoveRelative(Distance := rDistanceByVol[8], Velocity := aVelocity[8], Acc := aVelocity[8], Dec := aVelocity[8]);
END_IF
IF bMoveDistancePumps[9] THEN
	bMoveDistancePumps[9] := NOT GVL_Motion.aPumpsRotary[9].MoveRelative(Distance := rDistanceByVol[9], Velocity := aVelocity[9], Acc := aVelocity[9], Dec := aVelocity[9]);
END_IF
IF bMoveDistancePumps[10] THEN
	bMoveDistancePumps[10] := NOT GVL_Motion.aPumpsRotary[10].MoveRelative(Distance := rDistanceByVol[10], Velocity := aVelocity[10], Acc := aVelocity[10], Dec := aVelocity[10]);
END_IF

IF NOT bMoveDistancePumps[1] AND NOT bMoveDistancePumps[2] AND NOT bMoveDistancePumps[3] AND NOT bMoveDistancePumps[4] AND NOT bMoveDistancePumps[5] AND NOT bMoveDistancePumps[6] AND NOT bMoveDistancePumps[7] AND NOT bMoveDistancePumps[8] AND NOT bMoveDistancePumps[9] AND NOT bMoveDistancePumps[10] THEN
	bRequestMoveByDistance := FALSE;
	MoveByDistance := TRUE;
	RETURN;
ELSE
	MoveByDistance := FALSE;
END_IF
END_METHOD

METHOD MoveBySpeed : BOOL
VAR_INPUT
	aPumpIds		: ARRAY[1..10] OF BOOL;
	aPumpDirection 	: ARRAY[1..10] OF E_PumpDirection;
	aVelocity 		: ARRAY[1..10] OF REAL;
END_VAR
IF NOT bRequestMoveBySpeed THEN
	MoveBySpeed := FALSE;
	bMoveVelocityPumps := aPumpIds;
	bRequestMoveBySpeed := TRUE;
END_IF

IF bMoveVelocityPumps[1] THEN
	bMoveVelocityPumps[1] := NOT GVL_Motion.aPumpsRotary[1].MoveVelocity(rVelocity := aVelocity[1], rAcc := aVelocity[1], rDec := aVelocity[1], iDirection := aPumpDirection[1]);
END_IF
IF bMoveVelocityPumps[2] THEN
	bMoveVelocityPumps[2] := NOT GVL_Motion.aPumpsRotary[2].MoveVelocity(rVelocity := aVelocity[2], rAcc := aVelocity[2], rDec := aVelocity[2], iDirection := aPumpDirection[2]);
END_IF
IF bMoveVelocityPumps[3] THEN
	bMoveVelocityPumps[3] := NOT GVL_Motion.aPumpsRotary[3].MoveVelocity(rVelocity := aVelocity[3], rAcc := aVelocity[3], rDec := aVelocity[3], iDirection := aPumpDirection[3]);
END_IF
IF bMoveVelocityPumps[4] THEN
	bMoveVelocityPumps[4] := NOT GVL_Motion.aPumpsRotary[4].MoveVelocity(rVelocity := aVelocity[4], rAcc := aVelocity[4], rDec := aVelocity[4], iDirection := aPumpDirection[4]);
END_IF
IF bMoveVelocityPumps[5] THEN
	bMoveVelocityPumps[5] := NOT GVL_Motion.aPumpsRotary[5].MoveVelocity(rVelocity := aVelocity[5], rAcc := aVelocity[5], rDec := aVelocity[5], iDirection := aPumpDirection[5]);
END_IF
IF bMoveVelocityPumps[6] THEN
	bMoveVelocityPumps[6] := NOT GVL_Motion.aPumpsRotary[6].MoveVelocity(rVelocity := aVelocity[6], rAcc := aVelocity[6], rDec := aVelocity[6], iDirection := aPumpDirection[6]);
END_IF
IF bMoveVelocityPumps[7] THEN
	bMoveVelocityPumps[7] := NOT GVL_Motion.aPumpsRotary[7].MoveVelocity(rVelocity := aVelocity[7], rAcc := aVelocity[7], rDec := aVelocity[7], iDirection := aPumpDirection[7]);
END_IF
IF bMoveVelocityPumps[8] THEN
	bMoveVelocityPumps[8] := NOT GVL_Motion.aPumpsRotary[8].MoveVelocity(rVelocity := aVelocity[8], rAcc := aVelocity[8], rDec := aVelocity[8], iDirection := aPumpDirection[8]);
END_IF
IF bMoveVelocityPumps[9] THEN
	bMoveVelocityPumps[9] := NOT GVL_Motion.aPumpsRotary[9].MoveVelocity(rVelocity := aVelocity[9], rAcc := aVelocity[9], rDec := aVelocity[9], iDirection := aPumpDirection[9]);
END_IF
IF bMoveVelocityPumps[10] THEN
	bMoveVelocityPumps[10] := NOT GVL_Motion.aPumpsRotary[10].MoveVelocity(rVelocity := aVelocity[10], rAcc := aVelocity[10], rDec := aVelocity[10], iDirection := aPumpDirection[10]);
END_IF

IF NOT bMoveVelocityPumps[1] AND NOT bMoveVelocityPumps[2] AND NOT bMoveVelocityPumps[3] AND NOT bMoveVelocityPumps[4] AND NOT bMoveVelocityPumps[5] AND NOT bMoveVelocityPumps[6] AND NOT bMoveVelocityPumps[7] AND NOT bMoveVelocityPumps[8] AND NOT bMoveVelocityPumps[9] AND NOT bMoveVelocityPumps[10] THEN
	bRequestMoveBySpeed := FALSE;
	MoveBySpeed := TRUE;
	RETURN;
ELSE
	MoveBySpeed := FALSE;
END_IF
END_METHOD

METHOD MoveByVolume : BOOL
VAR_INPUT
	aPumpIds		: ARRAY[1..10] OF BOOL;
	aVolume 		: ARRAY[1..10] OF REAL;
	aPumpDirection 	: ARRAY[1..10] OF E_PumpDirection;
	aVelocity	 	: ARRAY[1..10] OF REAL;
END_VAR
VAR 
END_VAR
IF NOT bRequestMoveByVol THEN
	MoveByVolume := FALSE;
	bMoveRelativePumps := aPumpIds;
	bRequestMoveByVol := TRUE;
END_IF

//getting the valves position
aValvePosition[1] := F_GetValvePosition(iValveIndex := 1);
aValvePosition[2] := F_GetValvePosition(iValveIndex := 1);
aValvePosition[3] := F_GetValvePosition(iValveIndex := 2);
aValvePosition[4] := F_GetValvePosition(iValveIndex := 2);
aValvePosition[5] := F_GetValvePosition(iValveIndex := 3);
aValvePosition[6] := F_GetValvePosition(iValveIndex := 3);
aValvePosition[7] := F_GetValvePosition(iValveIndex := 4);
aValvePosition[8] := F_GetValvePosition(iValveIndex := 4);
aValvePosition[9] := F_GetValvePosition(iValveIndex := 5);
aValvePosition[10] := F_GetValvePosition(iValveIndex := 5);

//getting the pump factor based on pump path
aPumpPath[1] := F_GetPumpPath( iValvePosition := aValvePosition[1], ePumpDirection := aPumpDirection[1]);
aPumpPath[2] := F_GetPumpPath( iValvePosition := aValvePosition[2], ePumpDirection := aPumpDirection[2]);
aPumpPath[3] := F_GetPumpPath( iValvePosition := aValvePosition[3], ePumpDirection := aPumpDirection[3]);
aPumpPath[4] := F_GetPumpPath( iValvePosition := aValvePosition[4], ePumpDirection := aPumpDirection[4]);
aPumpPath[5] := F_GetPumpPath( iValvePosition := aValvePosition[5], ePumpDirection := aPumpDirection[5]);
aPumpPath[6] := F_GetPumpPath( iValvePosition := aValvePosition[6], ePumpDirection := aPumpDirection[6]);
aPumpPath[7] := F_GetPumpPath( iValvePosition := aValvePosition[7], ePumpDirection := aPumpDirection[7]);
aPumpPath[8] := F_GetPumpPath( iValvePosition := aValvePosition[8], ePumpDirection := aPumpDirection[8]);
aPumpPath[9] := F_GetPumpPath( iValvePosition := aValvePosition[9], ePumpDirection := aPumpDirection[9]);
aPumpPath[10] := F_GetPumpPath( iValvePosition := aValvePosition[10], ePumpDirection := aPumpDirection[10]);

//getting pump factor in mL/rev and converting to uL/degrees.
rDistanceByVol[1] := F_VolumeToSteps_Path(rVolume := aVolume[1], iPumpIndex := 1, ePath :=  aPumpPath[1]);
rDistanceByVol[2] := F_VolumeToSteps_Path(rVolume := aVolume[2], iPumpIndex := 2, ePath :=  aPumpPath[2]);
rDistanceByVol[3] := F_VolumeToSteps_Path(rVolume := aVolume[3], iPumpIndex := 3, ePath :=  aPumpPath[3]);
rDistanceByVol[4] := F_VolumeToSteps_Path(rVolume := aVolume[4], iPumpIndex := 4, ePath :=  aPumpPath[4]);
rDistanceByVol[5] := F_VolumeToSteps_Path(rVolume := aVolume[5], iPumpIndex := 5, ePath :=  aPumpPath[5]);
rDistanceByVol[6] := F_VolumeToSteps_Path(rVolume := aVolume[6], iPumpIndex := 6, ePath :=  aPumpPath[6]);
rDistanceByVol[7] := F_VolumeToSteps_Path(rVolume := aVolume[7], iPumpIndex := 7, ePath :=  aPumpPath[7]);
rDistanceByVol[8] := F_VolumeToSteps_Path(rVolume := aVolume[8], iPumpIndex := 8, ePath :=  aPumpPath[8]);
rDistanceByVol[9] := F_VolumeToSteps_Path(rVolume := aVolume[9], iPumpIndex := 9, ePath :=  aPumpPath[9]);
rDistanceByVol[10] := F_VolumeToSteps_Path(rVolume := aVolume[10], iPumpIndex := 10, ePath :=  aPumpPath[10]);



//Inverting the distance based on pumps flow direction
IF aPumpDirection[1] = E_PumpDirection.Backward THEN
	rDistanceByVol[1] := rDistanceByVol[1] * -1;
END_IF
IF aPumpDirection[2] = E_PumpDirection.Backward THEN
	rDistanceByVol[2] := rDistanceByVol[2] * -1;
END_IF
IF aPumpDirection[3] = E_PumpDirection.Backward THEN
	rDistanceByVol[3] := rDistanceByVol[3] * -1;
END_IF
IF aPumpDirection[4] = E_PumpDirection.Backward THEN
	rDistanceByVol[4] := rDistanceByVol[4] * -1;
END_IF
IF aPumpDirection[5] = E_PumpDirection.Backward THEN
	rDistanceByVol[5] := rDistanceByVol[5] * -1;
END_IF
IF aPumpDirection[6] = E_PumpDirection.Backward THEN
	rDistanceByVol[6] := rDistanceByVol[6] * -1;
END_IF
IF aPumpDirection[7] = E_PumpDirection.Backward THEN
	rDistanceByVol[7] := rDistanceByVol[7] * -1;
END_IF
IF aPumpDirection[8] = E_PumpDirection.Backward THEN
	rDistanceByVol[8] := rDistanceByVol[8] * -1;
END_IF
IF aPumpDirection[9] = E_PumpDirection.Backward THEN
	rDistanceByVol[9] := rDistanceByVol[9] * -1;
END_IF
IF aPumpDirection[10] = E_PumpDirection.Backward THEN
	rDistanceByVol[10] := rDistanceByVol[10] * -1;
END_IF

//Pumps relative movement
IF bMoveRelativePumps[1] THEN
	bMoveRelativePumps[1] := NOT GVL_Motion.aPumpsRotary[1].MoveRelative(Distance := rDistanceByVol[1], Velocity := aVelocity[1], Acc := aVelocity[1], Dec := aVelocity[1]);
END_IF
IF bMoveRelativePumps[2] THEN
	bMoveRelativePumps[2] := NOT GVL_Motion.aPumpsRotary[2].MoveRelative(Distance := rDistanceByVol[2], Velocity := aVelocity[2], Acc := aVelocity[2], Dec := aVelocity[2]);
END_IF
IF bMoveRelativePumps[3] THEN
	bMoveRelativePumps[3] := NOT GVL_Motion.aPumpsRotary[3].MoveRelative(Distance := rDistanceByVol[3], Velocity := aVelocity[3], Acc := aVelocity[3], Dec := aVelocity[3]);
END_IF
IF bMoveRelativePumps[4] THEN
	bMoveRelativePumps[4] := NOT GVL_Motion.aPumpsRotary[4].MoveRelative(Distance := rDistanceByVol[4], Velocity := aVelocity[4], Acc := aVelocity[4], Dec := aVelocity[4]);
END_IF
IF bMoveRelativePumps[5] THEN
	bMoveRelativePumps[5] := NOT GVL_Motion.aPumpsRotary[5].MoveRelative(Distance := rDistanceByVol[5], Velocity := aVelocity[5], Acc := aVelocity[5], Dec := aVelocity[5]);
END_IF
IF bMoveRelativePumps[6] THEN
	bMoveRelativePumps[6] := NOT GVL_Motion.aPumpsRotary[6].MoveRelative(Distance := rDistanceByVol[6], Velocity := aVelocity[6], Acc := aVelocity[6], Dec := aVelocity[6]);
END_IF
IF bMoveRelativePumps[7] THEN
	bMoveRelativePumps[7] := NOT GVL_Motion.aPumpsRotary[7].MoveRelative(Distance := rDistanceByVol[7], Velocity := aVelocity[7], Acc := aVelocity[7], Dec := aVelocity[7]);
END_IF
IF bMoveRelativePumps[8] THEN
	bMoveRelativePumps[8] := NOT GVL_Motion.aPumpsRotary[8].MoveRelative(Distance := rDistanceByVol[8], Velocity := aVelocity[8], Acc := aVelocity[8], Dec := aVelocity[8]);
END_IF
IF bMoveRelativePumps[9] THEN
	bMoveRelativePumps[9] := NOT GVL_Motion.aPumpsRotary[9].MoveRelative(Distance := rDistanceByVol[9], Velocity := aVelocity[9], Acc := aVelocity[9], Dec := aVelocity[9]);
END_IF
IF bMoveRelativePumps[10] THEN
	bMoveRelativePumps[10] := NOT GVL_Motion.aPumpsRotary[10].MoveRelative(Distance := rDistanceByVol[10], Velocity := aVelocity[10], Acc := aVelocity[10], Dec := aVelocity[10]);
END_IF

IF NOT bMoveRelativePumps[1] AND NOT bMoveRelativePumps[2] AND NOT bMoveRelativePumps[3] AND NOT bMoveRelativePumps[4] AND NOT bMoveRelativePumps[5] AND NOT bMoveRelativePumps[6] AND NOT bMoveRelativePumps[7] AND NOT bMoveRelativePumps[8] AND NOT bMoveRelativePumps[9] AND NOT bMoveRelativePumps[10] THEN
	bRequestMoveByVol := FALSE;
	MoveByVolume := TRUE;
	RETURN;
ELSE
	MoveByVolume := FALSE;
END_IF
END_METHOD

METHOD MoveLinearPumps : BOOL
VAR_INPUT
END_VAR
END_METHOD

METHOD Reset : BOOL
VAR_INPUT
END_VAR
VAR
    i : INT;
END_VAR
// ============================================================================
// FB_AllPumpsController.Reset()
// ---------------------------------------------------------------------------
// Logic reset only:
// - Clears all pending requests (MoveBySpeed/Vol/Distance/Linear + StopAllPumps)
// - Clears all internal "one-shot" arrays (move/stop flags)
// - Clears cached helper arrays (distance, valve positions, path)
// - Does NOT stop axes by itself (unless you decide to call StopAllPumps separately)
// ============================================================================

Reset := FALSE;

// 1) Clear pending "request" latches
bRequestMoveBySpeed     := FALSE;
bRequestMoveByVol       := FALSE;
bRequestMoveByDistance  := FALSE;
bRequestMoveLinearPumps := FALSE;
bRequestStopAllPumps    := FALSE;

// 2) Clear internal command arrays
FOR i := 1 TO 10 DO
    bMoveVelocityPumps[i] := FALSE;
    bMoveDistancePumps[i] := FALSE;
    bMoveRelativePumps[i] := FALSE;
    bMoveLinearPumps[i]   := FALSE;

    bStopRotaryPump[i] := FALSE;
    bStopLinearPump[i] := FALSE;

    // Helper/cached arrays (optional but recommended)
    rDistanceByVol[i] := 0.0;
    aValvePosition[i] := 0;
    aPumpPath[i]      := E_PumpPath.FillCalBox; // adjust if your enum has a proper "default"
END_FOR

Reset := TRUE;
END_METHOD

METHOD StopAllPumps : BOOL
VAR_INPUT
END_VAR
VAR
    i        : INT;
    bAllDone : BOOL;
END_VAR
// Default output
StopAllPumps := FALSE;

// ======================================================================
// 1) First trigger: prepare Stop request for ALL pumps
// ======================================================================
IF NOT bRequestStopAllPumps THEN
    StopAllPumps := FALSE;

    // Cancel any pending movement requests coming from this FB
    bRequestMoveBySpeed     := FALSE;
    bRequestMoveByVol       := FALSE;
    bRequestMoveByDistance  := FALSE;
    bRequestMoveLinearPumps := FALSE;

    // Clear internal movement arrays (to avoid Move + Stop clash)
    FOR i := 1 TO 10 DO
        bMoveVelocityPumps[i] := FALSE;
        bMoveDistancePumps[i] := FALSE;
        bMoveRelativePumps[i] := FALSE;
        bMoveLinearPumps[i]   := FALSE;

        // Set stop request for all rotary pumps
        bStopRotaryPump[i] := TRUE;

        // If linear pumps also have a stop method, prepare here:
        // bStopLinearPump[i] := TRUE;
    END_FOR

    bRequestStopAllPumps := TRUE;
END_IF

// ======================================================================
// 2) Execute Stop() for each pump that still requires stopping
// ======================================================================
FOR i := 1 TO 10 DO
    IF bStopRotaryPump[i] THEN
        // Call the Stop() method of the rotary pump i
        IF GVL_Motion.aPumpsRotary[i].Stop() THEN
            // When Stop() returns TRUE once, it means the pump has fully stopped
            bStopRotaryPump[i] := FALSE;
        END_IF
    END_IF
END_FOR

// ======================================================================
// 3) Check if ALL pumps have finished their Stop()
// ======================================================================
bAllDone := TRUE;

FOR i := 1 TO 10 DO
    IF bStopRotaryPump[i] THEN
        bAllDone := FALSE;
    END_IF
END_FOR

// ======================================================================
// 4) If all pumps are done, return TRUE once and reset internal flags
// ======================================================================
IF bAllDone THEN
    bRequestStopAllPumps := FALSE;
    StopAllPumps := TRUE;   // one pulse when everything is stopped
ELSE
    StopAllPumps := FALSE;
END_IF


(* Before Nov21 2025 --------------------------------------------------------------------------------------------------------------------------------------------------------------------------
IF NOT bRequestStopAllPumps THEN
	StopAllPumps := FALSE;
	bStopRotaryPump[1] := TRUE;
	bStopRotaryPump[2] := TRUE;
	bStopRotaryPump[3] := TRUE;
	bStopRotaryPump[4] := TRUE;
	bStopRotaryPump[5] := TRUE;
	bStopRotaryPump[6] := TRUE;
	bStopRotaryPump[7] := TRUE;
	bStopRotaryPump[8] := TRUE;
	bStopRotaryPump[9] := TRUE;
	bStopRotaryPump[10] := TRUE;
	bRequestStopAllPumps := TRUE;
END_IF

IF bStopRotaryPump[1] THEN
	bStopRotaryPump[1] := NOT GVL_Motion.aPumpsRotary[1].Stop();
END_IF
IF bStopRotaryPump[2] THEN
	bStopRotaryPump[2] := NOT GVL_Motion.aPumpsRotary[2].Stop();
END_IF
IF bStopRotaryPump[3] THEN
	bStopRotaryPump[3] := NOT GVL_Motion.aPumpsRotary[3].Stop();
END_IF
IF bStopRotaryPump[4] THEN
	bStopRotaryPump[4] := NOT GVL_Motion.aPumpsRotary[4].Stop();
END_IF
IF bStopRotaryPump[5] THEN
	bStopRotaryPump[5] := NOT GVL_Motion.aPumpsRotary[5].Stop();
END_IF
IF bStopRotaryPump[6] THEN
	bStopRotaryPump[6] := NOT GVL_Motion.aPumpsRotary[6].Stop();
END_IF
IF bStopRotaryPump[7] THEN
	bStopRotaryPump[7] := NOT GVL_Motion.aPumpsRotary[7].Stop();
END_IF
IF bStopRotaryPump[8] THEN
	bStopRotaryPump[8] := NOT GVL_Motion.aPumpsRotary[8].Stop();
END_IF
IF bStopRotaryPump[9] THEN
	bStopRotaryPump[9] := NOT GVL_Motion.aPumpsRotary[9].Stop();
END_IF
IF bStopRotaryPump[10] THEN
	bStopRotaryPump[10] := NOT GVL_Motion.aPumpsRotary[10].Stop();
END_IF

IF NOT bStopRotaryPump[1] AND NOT bStopRotaryPump[2] AND NOT bStopRotaryPump[3] AND NOT bStopRotaryPump[4] AND NOT bStopRotaryPump[5] AND NOT bStopRotaryPump[6] AND NOT bStopRotaryPump[7] AND NOT bStopRotaryPump[8] AND NOT bStopRotaryPump[9] AND NOT bStopRotaryPump[10] THEN
	bRequestStopAllPumps := FALSE;
	StopAllPumps := TRUE;
	RETURN;
ELSE
	StopAllPumps := FALSE;
END_IF
*)
END_METHOD

END_FUNCTION_BLOCK

// ---- POUs/Functions/F_GetValvePosition.TcPOU
FUNCTION F_GetValvePosition : SINT
VAR_INPUT
	iValveIndex	: USINT; // Valve index
END_VAR
VAR
	rValveActualPos		: LREAL; // valve actual position
	rPositionTolerance	: REAL := 2.0;
END_VAR

//Funtion to get the actual valve position
rValveActualPos := GVL_Motion.aValves[iValveIndex].rActualPos;

IF rValveActualPos > 0 - rPositionTolerance AND rValveActualPos < 0 + rPositionTolerance THEN
	F_GetValvePosition := 1;
	RETURN;
END_IF

IF rValveActualPos > 1200 - rPositionTolerance AND rValveActualPos < 1200 + rPositionTolerance THEN
	F_GetValvePosition := 2;
	RETURN;
END_IF

IF rValveActualPos > 2400 - rPositionTolerance AND rValveActualPos < 2400 + rPositionTolerance THEN
	F_GetValvePosition := 3;
	RETURN;
END_IF

IF rValveActualPos > 3600 - rPositionTolerance AND rValveActualPos < 3600 + rPositionTolerance THEN
	F_GetValvePosition := 4;
	RETURN;
END_IF

IF rValveActualPos > 4800 - rPositionTolerance AND rValveActualPos < 4800 + rPositionTolerance THEN
	F_GetValvePosition := 5;
	RETURN;
END_IF

IF rValveActualPos > 6000 - rPositionTolerance AND rValveActualPos < 6000 + rPositionTolerance THEN
	F_GetValvePosition := 6;
	RETURN;
END_IF

F_GetValvePosition := -1;
RETURN;

END_FUNCTION

// ---- POUs/Functions/F_GetPumpPath.TcPOU
FUNCTION F_GetPumpPath : E_PumpPath
VAR_INPUT
	iValvePosition	: SINT;
	ePumpDirection	: E_PumpDirection;
END_VAR
VAR
END_VAR

CASE iValvePosition OF
	
	1:
		F_GetPumpPath := E_PumpPath.FillJars;
		RETURN;
	
	2:
		F_GetPumpPath := E_PumpPath.FillJars;
		RETURN;
	
	3:
		F_GetPumpPath := E_PumpPath.FillJars;
		RETURN;
		
	4:
		F_GetPumpPath := E_PumpPath.FillJars;
		RETURN;
		
	5:
		F_GetPumpPath := E_PumpPath.FillCalBox;
		RETURN;
	6:
		IF ePumpDirection = E_PumpDirection.Forward THEN
			F_GetPumpPath := E_PumpPath.FromCalBox;
			RETURN;
			ELSIF ePumpDirection = E_PumpDirection.Backward THEN
				F_GetPumpPath := E_PumpPath.FillCalBox;
				RETURN;
		ELSE
			F_GetPumpPath := E_PumpPath.FromCalBox;
			RETURN;
		END_IF

END_CASE

END_FUNCTION

// ---- POUs/Functions/F_JarName.TcPOU
FUNCTION F_JarName : STRING
VAR_INPUT
	iPumpIndex : UINT;
END_VAR
VAR
END_VAR

CASE iPumpIndex OF
	1: F_JarName := 'T/C'; RETURN;
	2: F_JarName := 'S0'; RETURN;
	3: F_JarName := 'S1'; RETURN;
	4: F_JarName := 'S2'; RETURN;
	5: F_JarName := 'S3'; RETURN;
	6: F_JarName := 'S4'; RETURN;
	7: F_JarName := 'S5'; RETURN;
	8: F_JarName := 'S6'; RETURN;
	9: F_JarName := 'S7'; RETURN;
	10: F_JarName := 'F'; RETURN;
ELSE
	F_JarName := ''; RETURN;
END_CASE

END_FUNCTION

// ---- POUs/Functions/F_sec_to_time.TcPOU
FUNCTION F_sec_to_time : TIME
VAR_INPUT
	sec : LREAL;
END_VAR
VAR
END_VAR

F_sec_to_time := LREAL_TO_TIME(MAX(0.0, sec) * 1000.0);

END_FUNCTION

// ---- POUs/5. Calibration/FB_SaveCalibrationReport.TcPOU
(*
    FB_SaveCalibrationReport
    - One-shot wrapper: builds the calibration JSON and writes it to disk.
*)
FUNCTION_BLOCK FB_SaveCalibrationReport
VAR_INPUT
	bExecute            : BOOL;  // Rising edge starts the build+save sequence
    sUser               : STRING(64);

    stReportInfo        : ST_ReportInfo;
    stCalibrationInfo   : ST_CalibrationInfo;
    aCalibrationData    : ARRAY[1..250] OF ST_CalibrationData;
    iDataCount          : INT;   // Valid range: 0..100 (0 allowed -> empty list)
END_VAR
VAR_OUTPUT
	bDone       : BOOL;          // TRUE when file is saved and closed
    bBusy       : BOOL;          // TRUE while internal state machine is running
    bError      : BOOL;          // TRUE on any error
    nErrId      : UDINT;         // Error code propagated from child FBs
    sFileNameOut: STRING(256);   // Full path of the output JSON file
END_VAR
VAR
	// State machine
    iStep       : INT;           // 0=IDLE, 10=BUILD, 20=SAVE, 100=LATCH

    // Edge detection for bExecute
    rtExec      : R_TRIG;

    // Child FBs
    fbBuild     : FB_BuildCalReportJson;
    fbSave      : FB_SaveCalReportToFile;

    // Buffer for JSON document produced by builder
    sBuf        : STRING(16384);
	nBufBytes 	: UDINT;          // <- NEW
END_VAR

// --------------------------- IMPLEMENTATION ----------------------------------
rtExec(CLK := bExecute);

CASE iStep OF
    // -------------------------------------------------------------------------
    0: // IDLE: arm on rising edge of bExecute
    // -------------------------------------------------------------------------
    IF rtExec.Q THEN
        // Clamp iDataCount to valid limits (defensive)
        IF iDataCount < 0   THEN iDataCount := 0;   END_IF;
        IF iDataCount > 100 THEN iDataCount := 100; END_IF;

        // Clear latched outputs and mark busy
        bDone := FALSE; bError := FALSE; nErrId := 0;
        sFileNameOut := '';
        bBusy := TRUE;

        // Jump to build step
        iStep := 10;
    END_IF

    // -------------------------------------------------------------------------
    10: // BUILD JSON: FB_BuildCalReportJson (single-shot)
    // -------------------------------------------------------------------------
    fbBuild(
        stReportInfo      := stReportInfo,
        stCalibrationInfo := stCalibrationInfo,
        aCalibrationData  := aCalibrationData,
		iCalNumber  	  := TO_INT(stCalibrationInfo.iCalibrationNumber),
		sUser        	  := sUser,
        iDataCount        := iDataCount
    );

    IF fbBuild.bDone THEN
        // Copy the produced JSON document into our local buffer
        sBuf      := fbBuild.sJsonBuffer;
		nBufBytes := fbBuild.nJsonBytes;
		sFileNameOut := fbBuild.sFileNameOut;

        // Proceed to SAVE step
        iStep := 20;

    ELSIF fbBuild.bError THEN
        // Propagate error and latch
        bError := TRUE;
        nErrId := fbBuild.nErrId;
        bBusy := FALSE;
        iStep := 100;
    END_IF

    // -------------------------------------------------------------------------
    20: // SAVE FILE: FB_SaveCalReportToFile (stateful)
    // -------------------------------------------------------------------------
    
	fbSave(
        bExecute    := TRUE,  // keep TRUE while we wait for bDone/bError
        sJsonBuffer := sBuf,
		nJsonBytes  := nBufBytes,
		sFileNameIn := sFileNameOut,
    );

    IF fbSave.bDone THEN
        bDone := TRUE;
        bBusy := FALSE;
        iStep := 100;

    ELSIF fbSave.bError THEN
        bError := TRUE;
        nErrId := fbSave.nErrId;
        bBusy := FALSE;
        iStep := 100;
    END_IF

    // -------------------------------------------------------------------------
    100: // LATCH: wait caller to drop bExecute to return to IDLE
    // -------------------------------------------------------------------------
    // Keep driving fbSave with bExecute := FALSE to let it reset internally.
    fbSave(bExecute := FALSE);

    IF NOT bExecute THEN
        // Return to IDLE after caller drops the trigger
        iStep := 0;
    END_IF
END_CASE

METHOD Reset : BOOL
VAR_INPUT
END_VAR
// Latch outputs & codes
bDone        := FALSE;
bBusy        := FALSE;
bError       := FALSE;
nErrId       := 0;
sFileNameOut := '';

// State machine
iStep := 0;

// Internal buffers
sBuf      := '';
nBufBytes := 0;

// Politely reset child FBs (if their Reset() exists; otherwise just de-assert)
fbBuild.Reset(); // returns TRUE/ignored; leaves builder idle
fbSave.Reset();  // returns TRUE/ignored; leaves saver idle

// Extra safety: ensure no lingering executes this cycle
fbSave(bExecute := FALSE);

Reset := TRUE;
END_METHOD

END_FUNCTION_BLOCK

// ---- POUs/5. Calibration/FB_BuildCalReportJson.TcPOU
(*
    FB_BuildCalReportJson
    - Gera o JSON do relatório de calibração em sJsonBuffer (sem gravar em disco).
    - Alinhado ao schema do reportASRS.json.
*)
FUNCTION_BLOCK FB_BuildCalReportJson
VAR_INPUT
	stReportInfo        : ST_ReportInfo;               			// GVL_Calibration.stPumpCalReportInfo
    stCalibrationInfo   : ST_CalibrationInfo;          			// GVL_Calibration.stPumpCalibrationInfo
    aCalibrationData    : ARRAY[1..250] OF ST_CalibrationData; 	// GVL_Calibration.stPumpCalibrationData
    iDataCount          : INT;                         			// Quantos itens válidos em aCalibrationData (1..100)
	sUser       		: STRING(64);							// Username used in file name
	iCalNumber  		: INT;                  				// Calibration number used in file name
END_VAR
VAR_OUTPUT
	bDone       : BOOL;
    bBusy       : BOOL;
    bError      : BOOL;
    nErrId      : UDINT;
    sJsonBuffer : STRING(32767);
	nJsonBytes  : UDINT;  // exact byte count (excludes trailing #0)
	sFileNameOut: STRING(256); 
END_VAR
VAR
	fbJson          : FB_JsonDomParser;
    rootObj         : SJsonValue;
    objRepInfo      : SJsonValue;
    objCalInfo      : SJsonValue;
    arrCalData      : SJsonValue;
    rowObj          : SJsonValue;

    i               : INT;
    sTmp            : STRING(256);
    sY              : STRING(4);
    sM              : STRING(2);
    sD              : STRING(2);
    sDateOnly       : STRING(16);
    sDateTimeOnly   : STRING(32);
    sTimeOnly       : STRING(16);
	nCopied 		: UDINT;
	
	// Timestamp generation (local system time)
	fbLocalSystemTime : FB_LocalSystemTime;
    stLocal           : TIMESTRUCT;
    sStamp            : STRING(32);
    sHH               : STRING(2);
    sMM               : STRING(2);
    sSS               : STRING(2);
    sMMo              : STRING(2);
    sDD               : STRING(2);
	bDTReady		  : BOOL := FALSE;
	
	// File name helpers
    sUserSafe       : STRING(64);
	sFileName		: STRING(256);
	
	bBuildStart		: BOOL := FALSE;
	
END_VAR

// ---------- Execução única ----------
bBusy := TRUE; bDone := FALSE; bError := FALSE; nErrId := 0;

// Garante limites
IF iDataCount < 0 THEN iDataCount := 0; END_IF
IF iDataCount > 100 THEN iDataCount := 100; END_IF

// Generates de File Name using the date  
// Produce a timestamp: YYYYMMDD_HHMMSS
fbLocalSystemTime(bEnable := TRUE, dwCycle := 5);
IF fbLocalSystemTime.bValid THEN
	stLocal := fbLocalSystemTime.systemTime;

	sMMo := F_TwoDigits(stLocal.wMonth);
	sDD  := F_TwoDigits(stLocal.wDay);
	sHH  := F_TwoDigits(stLocal.wHour);
	sMM  := F_TwoDigits(stLocal.wMinute);
	sSS  := F_TwoDigits(stLocal.wSecond);

	sStamp := CONCAT(INT_TO_STRING(stLocal.wYear), sMMo);       // YYYYMM
	sStamp := CONCAT(sStamp, sDD);                              // YYYYMMDD
	sStamp := CONCAT(sStamp, '_');                              // YYYYMMDD_
	sStamp := CONCAT(sStamp, sHH);                              // YYYYMMDD_HH
	sStamp := CONCAT(sStamp, sMM);                              // YYYYMMDD_HHMM
	sStamp := CONCAT(sStamp, sSS);                              // YYYYMMDD_HHMMSS
	
	bDTReady := TRUE;
	
ELSE
	sStamp := '00000000_000000'; // Fallback if system time is not valid
END_IF

IF bDTReady THEN

	sUserSafe := sUser;

	// Build output file name
	sFileNameOut := CONCAT('C:/TwinCAT/Reports/PumpCalibration/',
					   CONCAT('Calib_', CONCAT(INT_TO_STRING(iCalNumber),
					   CONCAT('_', CONCAT(sUserSafe, CONCAT('_', CONCAT(sStamp, '.json')))))));
	
	// FileName going into JsonReport info 
	sFileName :=  CONCAT('Calib_', CONCAT(INT_TO_STRING(iCalNumber),
					   CONCAT('_', CONCAT(sUserSafe, CONCAT('_', sStamp)))));
	bDTReady := FALSE;
	bBuildStart := TRUE;
END_IF
IF bBuildStart THEN
	// Documento raiz
	rootObj := fbJson.NewDocument();
	
	// ===== reportInfo =====
	objRepInfo := fbJson.AddObjectMember(rootObj, 'reportInfo');
	fbJson.AddStringMember(objRepInfo, 'reportName',      stReportInfo.sReportName);
	fbJson.AddStringMember(objRepInfo, 'reoportSubName',  stReportInfo.sReoportSubName);
	fbJson.AddStringMember(objRepInfo, 'reportDate', stReportInfo.sReportDate);
	fbJson.AddStringMember(objRepInfo, 'systemID',     stReportInfo.sSystemID);
	fbJson.AddStringMember(objRepInfo, 'databaseName', stReportInfo.sDatabaseName);
	
	// iPage -> "02"
	sTmp := USINT_TO_STRING(stReportInfo.iPage);
	IF LEN(sTmp) = 1 THEN sTmp := CONCAT('0', sTmp); END_IF
	fbJson.AddStringMember(objRepInfo, 'page', sTmp);
	
	fbJson.AddStringMember(objRepInfo, 'printedBy', stReportInfo.sPrintedBy);
	fbJson.AddStringMember(objRepInfo, 'fileName', sFileName);
	
	// ===== calibrationInfo =====
	objCalInfo := fbJson.AddObjectMember(rootObj, 'parametersInfo');
	fbJson.AddIntMember(   objCalInfo, 'calibrationNumber', stCalibrationInfo.iCalibrationNumber);
	fbJson.AddStringMember(objCalInfo, 'userID',            stCalibrationInfo.iUserID);
	fbJson.AddDoubleMember(objCalInfo, 'density',           stCalibrationInfo.rSolventDensity);
	fbJson.AddStringMember(objCalInfo, 'solvent',           stCalibrationInfo.iSolventID);
	fbJson.AddIntMember(   objCalInfo, 'sysMasterListRev',  stCalibrationInfo.iSysMasterListRev);
	fbJson.AddIntMember(   objCalInfo, 'sysSetRev',  		stCalibrationInfo.iSysSettingsRev);
	fbJson.AddIntMember(   objCalInfo, 'solventRevision',   stCalibrationInfo.iSolventRevision);
	fbJson.AddIntMember(   objCalInfo, 'allowableFailures', stCalibrationInfo.iAllowableFailures);
	fbJson.AddIntMember(   objCalInfo, 'replicates',        stCalibrationInfo.iReplicates);
	fbJson.AddIntMember(   objCalInfo, 'calIntervalDays',   stCalibrationInfo.iCalIntervalDays);
		
	// ===== calibrationData (array de objetos) =====
	arrCalData := fbJson.AddArrayMember(rootObj, 'calibrationData', 0);
	
	FOR i := 1 TO iDataCount DO
		// Cria elemento no array e define como objeto		
		rowObj := fbJson.PushbackNullValue(arrCalData);
		fbJson.SetObject(rowObj);
		(*
		// Formata DT como "YYYY-MM-DD HH:MM:SS"
		sTmp := DT_TO_STRING(aCalibrationData[i].dDateTime); // "DT#YYYY-MM-DD-HH:MM:SS"
		IF LEFT(sTmp,3) = 'DT#' THEN
			sTmp := RIGHT(sTmp, LEN(sTmp)-3);                // "YYYY-MM-DD-HH:MM:SS"
		END_IF
		sDateOnly     := LEFT(sTmp, 10);                     // "YYYY-MM-DD"
		sTimeOnly     := RIGHT(sTmp, LEN(sTmp)-11);          // remove "YYYY-MM-DD-" (11 chars)
		sDateTimeOnly := CONCAT(sDateOnly, CONCAT(' ', sTimeOnly));
		*)
		fbJson.AddStringMember(rowObj, 'dateTime',             aCalibrationData[i].dDateTime);
		fbJson.AddIntMember(   rowObj, 'pumpNumber',           aCalibrationData[i].iPumpNumber);
		fbJson.AddStringMember(rowObj, 'step',                 aCalibrationData[i].sStep);
		fbJson.AddDoubleMember(rowObj, 'grossWt_g',            aCalibrationData[i].rGrossWeigth);
		fbJson.AddDoubleMember(rowObj, 'tareWt_g',             aCalibrationData[i].rTareWeigth);
		fbJson.AddDoubleMember(rowObj, 'netWt_g',              aCalibrationData[i].rNetWeigth);
		fbJson.AddDoubleMember(rowObj, 'netVolume',            aCalibrationData[i].rNetVolume);
		fbJson.AddDoubleMember(rowObj, 'targetVolume_ul',      aCalibrationData[i].rTargetVolume);
		fbJson.AddDoubleMember(rowObj, 'difference_ul',        aCalibrationData[i].rDifferenceUl);
		fbJson.AddDoubleMember(rowObj, 'difference_percent',   aCalibrationData[i].rDifferencePercent);
		fbJson.AddDoubleMember(rowObj, 'criteria',             aCalibrationData[i].rCriteria);
		fbJson.AddIntMember(   rowObj, 'pumpRev',              aCalibrationData[i].iPumpRevs);
	END_FOR
	
	// Serializa
	nCopied := fbJson.CopyDocument(sJsonBuffer, SIZEOF(sJsonBuffer));
	
	IF nCopied > 0 THEN
		nJsonBytes := nCopied - 1;  // remove terminator
		bDone := TRUE;
		bBuildStart := FALSE;
	ELSE
		bError := TRUE; nErrId := 16#CAFE0001;
		bBuildStart := FALSE;
	END_IF
	
	bBusy := FALSE;
	
END_IF

METHOD Reset : BOOL
VAR_INPUT
END_VAR
// Outputs
bDone        := FALSE;
bBusy        := FALSE;
bError       := FALSE;
nErrId       := 0;
sJsonBuffer  := '';
nJsonBytes   := 0;
sFileNameOut := '';

// Transient flags
bDTReady     := FALSE;
bBuildStart  := FALSE;

// JSON handles & locals
rootObj   := 0;
objRepInfo:= 0;
objCalInfo:= 0;
arrCalData:= 0;
rowObj    := 0;

nCopied   := 0;
i         := 0;

sTmp          := '';
sY            := '';
sM            := '';
sD            := '';
sDateOnly     := '';
sDateTimeOnly := '';
sTimeOnly     := '';

// Timestamp helpers & filename helpers
sStamp    := '';
sHH       := '';
sMM       := '';
sSS       := '';
sMMo      := '';
sDD       := '';
sUserSafe := '';
sFileName := '';

Reset := TRUE;
END_METHOD

END_FUNCTION_BLOCK

// ---- POUs/5. Calibration/FB_SaveCalReportToFile.TcPOU
(*
    FB_SaveCalReportToFile
    - Writes a JSON buffer to disk as a uniquely named file under:
        C:\TwinCAT\ReportsPumpCalibration\
    - File name pattern:
        Calib_<calibrationNumber>_<user>_<YYYYMMDD_HHMMSS>.json
*)
FUNCTION_BLOCK FB_SaveCalReportToFile
VAR_INPUT
	bExecute    : BOOL;                 // Rising edge starts the save sequence
    sJsonBuffer : STRING(16384);        // JSON payload to write (already built)
	nJsonBytes  : UDINT;        		// sJsonBuffer Lenght to create the file 
	sFileNameIn : STRING(256);			// File path used on file creation
END_VAR
VAR_OUTPUT
	bDone       : BOOL;                 // TRUE when file is fully written and closed
    bBusy       : BOOL;                 // TRUE while state machine is running
    bError      : BOOL;                 // TRUE on any error
    nErrId      : UDINT;                // Propagates underlying FB error code
END_VAR
VAR
	iStep           : INT;

    // File primitives (Tc2_Utilities)
    fbFileOpen      : FB_FileOpen;
    fbFileWrite     : FB_FileWrite;
    fbFileClose     : FB_FileClose;
    hFile           : UINT;
    nBytesToWrite   : UDINT;

    // Timestamp generation (local system time)
    fbLocalSystemTime : FB_LocalSystemTime;
    stLocal           : TIMESTRUCT;
    sStamp            : STRING(32);
    sHH               : STRING(2);
    sMM               : STRING(2);
    sSS               : STRING(2);
    sMMo              : STRING(2);
    sDD               : STRING(2);
	bDTReady		  : BOOL := FALSE;

    // File name helpers
    sUserSafe       : STRING(64);
	
	bCloseFileStart : BOOL := FALSE;
	
END_VAR

CASE iStep OF
    // -------------------------------------------------------------------------
    0: // Idle -> Arm
    // -------------------------------------------------------------------------
    IF bExecute THEN
        bBusy := TRUE; bDone := FALSE; bError := FALSE; nErrId := 0;

		iStep := 10;
    END_IF

    // -------------------------------------------------------------------------
    10: // Wait file open
    // -------------------------------------------------------------------------
	// Open (create/overwrite) file in TEXT mode
        fbFileOpen(
            sNetId   := '',
            sPathName:= sFileNameIn,
            nMode    := FOPEN_MODEWRITE OR FOPEN_MODETEXT,
            bExecute := TRUE
        );
        fbFileWrite(bExecute := FALSE);
        fbFileClose(bExecute := FALSE);
		
    IF NOT fbFileOpen.bBusy THEN
        IF fbFileOpen.bError THEN
            bError := TRUE; nErrId := fbFileOpen.nErrId;
            bBusy := FALSE; iStep := 100;
        ELSE
            hFile := fbFileOpen.hFile;
            iStep := 20;
        END_IF
    END_IF

    // -------------------------------------------------------------------------
    20: // Write JSON buffer
    // -------------------------------------------------------------------------

    // JSON already comes ready in sJsonBuffer; nJsonBytes gives number of characters
    nBytesToWrite := nJsonBytes;

    fbFileWrite(
        sNetId     := '',
        hFile      := hFile,
        pWriteBuff := ADR(sJsonBuffer),
        cbWriteLen := nBytesToWrite,
        bExecute   := TRUE
    );
    //iStep := 30;

    // -------------------------------------------------------------------------
    //30: // Wait write completion, then close
    // -------------------------------------------------------------------------
    IF NOT fbFileWrite.bBusy THEN
        IF fbFileWrite.bError THEN
            bError := TRUE; nErrId := fbFileWrite.nErrId;
            // Try closing handle even on error
			bCloseFileStart := TRUE;
            fbFileClose(sNetId := '', hFile := hFile, bExecute := TRUE);
        ELSE
            fbFileClose(sNetId := '', hFile := hFile, bExecute := TRUE);
			bCloseFileStart := TRUE;
        END_IF
    END_IF

    IF NOT fbFileClose.bBusy AND bCloseFileStart THEN
        IF fbFileClose.bError THEN
            bError := TRUE; nErrId := fbFileClose.nErrId;
        END_IF
        bDone := NOT bError;
        bBusy := FALSE;
        iStep := 100;
    END_IF

    // -------------------------------------------------------------------------
    100: // Latch until caller drops bExecute
    // -------------------------------------------------------------------------
    IF NOT bExecute THEN
        iStep := 0;
		bCloseFileStart := FALSE;
        bDone := FALSE; bBusy := FALSE; bError := FALSE; nErrId := 0;
    END_IF
END_CASE

METHOD Reset : BOOL
VAR_INPUT
END_VAR
// Best-effort close if a handle is present
IF hFile <> 0 THEN
    fbFileClose(sNetId := '', hFile := hFile, bExecute := TRUE);
END_IF;

// Ensure child file FBs are not executing
fbFileOpen(bExecute := FALSE);
fbFileWrite(bExecute := FALSE);
fbFileClose(bExecute := FALSE);

// Clear locals
hFile          := 0;
nBytesToWrite  := 0;
bCloseFileStart:= FALSE;

// Clear status & state
bDone := FALSE;
bBusy := FALSE;
bError:= FALSE;
nErrId:= 0;
iStep := 0;

Reset := TRUE;
END_METHOD

END_FUNCTION_BLOCK

// ---- POUs/Utilities/FB_DosingTest.TcPOU
FUNCTION_BLOCK FB_DosingTest
VAR_INPUT
 	iReplicate 		: USINT;
	bExecute		: BOOL;
	rVolumeTesting	: REAL;
	aPumps			: ARRAY[1..10] OF BOOL;
END_VAR
VAR_OUTPUT
	bDone 	: BOOL;
	bError 	: BOOL;
	bBusy 	: BOOL;
END_VAR
VAR
	eState 			: (Idle, MoveLinearMotors, MoveValvesSolvent, RunForward, MoveValveNeedles, RunBackwards, WeightRequest, NextPump, Done);
	rDistanceByVol	: ARRAY[1..10] OF LREAL;
	bValvesMove		: ARRAY[1..5]  OF BOOL;
	bPumpsMove		: BOOL;
	rScaleWeight	: LREAL;
	rWeightBefore	: LREAL;
	bWeightDone 	: BOOL := FALSE;
	bStartDosing	: BOOL := FALSE;
	bMoveMotorM3 	: BOOL := FALSE;
	bMoveMotorM2 	: BOOL := FALSE;
	
	RTrigExecutePulse   : R_TRIG;
	tonMotorsDelay		: TON;
	
	i			: USINT;
	iResults 	: USINT := 1;
	iResultRow	: USINT := 1;
	iPumpIndex	: USINT := 1;
	iRevs		: LREAL;

END_VAR

// Triggering pulse
RTrigExecutePulse(CLK := bExecute);

// FB Trigger
IF RTrigExecutePulse.Q AND eState = Idle THEN
    bStartDosing := TRUE;
END_IF

CASE eState OF

Idle:
    	bBusy := FALSE;
		bDone := FALSE;
		IF bStartDosing THEN
			iResults   := 1;
			iResultRow := 1;
			iPumpIndex := 1;
			rWeightBefore := 0;
			tonMotorsDelay(in := FALSE);
			bMoveMotorM2 := FALSE;
			bMoveMotorM3 := FALSE;
			bBusy  := TRUE;
			eState := MoveLinearMotors;
			bStartDosing := FALSE;
		END_IF
		
// Positioning Motors	
MoveLinearMotors:		
// Positioning motors M2 and M3 to calibration position 
		IF NOT bMoveMotorM3 THEN
			bMoveMotorM3 := GVL_Motion.aMotors[3].MoveAbsolute(GVL_Settings.stMachineParam.aM3Position[4], GVL_Settings.stMachineParam.rM3Velocity, GVL_Settings.stMachineParam.rM3Accleration, GVL_Settings.stMachineParam.rM3Deceleration);
		END_IF
		IF NOT bMoveMotorM2 AND bMoveMotorM3 THEN
			bMoveMotorM2 := GVL_Motion.aMotors[2].MoveAbsolute(GVL_Settings.stMachineParam.aM2Position[5], GVL_Settings.stMachineParam.rM2Velocity, GVL_Settings.stMachineParam.rM2Accleration, GVL_Settings.stMachineParam.rM2Deceleration);
		END_IF
	
		IF bMoveMotorM2 AND bMoveMotorM3 THEN
			tonMotorsDelay(in := TRUE, pt := T#200MS);
		END_IF
		
		IF tonMotorsDelay.Q THEN
			bMoveMotorM2 := FALSE;
			bMoveMotorM3 := FALSE;
			eState := MoveValvesSolvent;
		END_IF


// Positioning valves pos 1
MoveValvesSolvent:
	tonMotorsDelay(in := FALSE);
	FOR i := 1 TO 5 DO
		IF NOT bValvesMove[i] THEN
			bValvesMove[i] := GVL_Motion.aValvesObj[i].MoveValve(	iPosition := 1, 
																	rVelocity := GVL_Motion.aValves[i].rTargetVel, 
																	rAcc := GVL_Motion.aValves[i].rAcceleration, 
																	rDec := GVL_Motion.aValves[i].rDeceleration
																);
		END_IF
	END_FOR
	
	IF bValvesMove[1] AND bValvesMove[2] AND bValvesMove[3] AND bValvesMove[4] AND bValvesMove[5] THEN
		bPumpsMove := FALSE;
		eState := RunForward;
	END_IF
	

// pumps forward by volume
RunForward:
	
	IF NOT bMoveMotorM2 THEN
		bMoveMotorM2 := GVL_Motion.aMotors[2].MoveAbsolute(GVL_Settings.stMachineParam.aM2Position[5], GVL_Settings.stMachineParam.rM2Velocity, GVL_Settings.stMachineParam.rM2Accleration, GVL_Settings.stMachineParam.rM2Deceleration);
	END_IF

	IF bMoveMotorM2 THEN
		IF aPumps[iPumpIndex] THEN
			rDistanceByVol[iPumpIndex] := F_VolumeToSteps_Path(rVolume := rVolumeTesting + GVL_Motion.aPumps[iPumpIndex].Rotary.rDeadVolume, iPumpIndex := iPumpIndex, ePath := E_PumpPath.FromCalBox);
			
			iRevs := rDistanceByVol[iPumpIndex]/360;
			
			IF NOT bPumpsMove THEN
				bPumpsMove :=	GVL_Motion.aPumpsRotary[iPumpIndex].MoveRelative(	Distance := rDistanceByVol[iPumpIndex], 
																					Velocity := GVL_Settings.stPumpParameters.iMeterVelocity * 6,
																					Acc := GVL_Settings.stPumpParameters.iMeterVelocity * 6, 
																					Dec := GVL_Settings.stPumpParameters.iMeterVelocity * 6
																				);
			END_IF
		ELSE
			iPumpIndex := iPumpIndex + 1;
			//bPumpsMove := TRUE;
		END_IF
	END_IF
	
	IF bPumpsMove THEN
		FOR i := 1 TO 5 DO
			bValvesMove[i] := FALSE;
		END_FOR
		bMoveMotorM2 := FALSE; 
		eState := MoveValveNeedles;
	END_IF

// positioning valves pos6
MoveValveNeedles:
	FOR i := 1 TO 5 DO
		IF NOT bValvesMove[i] THEN
			bValvesMove[i] := GVL_Motion.aValvesObj[i].MoveValve(	iPosition := 6, 
																	rVelocity := GVL_Motion.aValves[i].rTargetVel, 
																	rAcc := GVL_Motion.aValves[i].rAcceleration, 
																	rDec := GVL_Motion.aValves[i].rDeceleration
																);
		END_IF
	END_FOR
	
	IF bValvesMove[1] AND bValvesMove[2] AND bValvesMove[3] AND bValvesMove[4] AND bValvesMove[5] THEN
		bPumpsMove := FALSE;
		eState := RunBackwards;
	END_IF

// pumps backward by volume
RunBackwards:
	IF aPumps[iPumpIndex] THEN
		
			rDistanceByVol[iPumpIndex] := F_VolumeToSteps_Path(rVolume := (rVolumeTesting + GVL_Motion.aPumps[iPumpIndex].Rotary.rDeadVolume) * 1.6, iPumpIndex := iPumpIndex, ePath := E_PumpPath.FromCalBox);
			
			IF NOT bPumpsMove THEN
				bPumpsMove := GVL_Motion.aPumpsRotary[iPumpIndex].MoveRelative(		Distance := - rDistanceByVol[iPumpIndex], 
																					Velocity := GVL_Settings.stPumpParameters.iMeterVelocity * 6,
																					Acc := GVL_Settings.stPumpParameters.iMeterVelocity * 6, 
																					Dec := GVL_Settings.stPumpParameters.iMeterVelocity * 6
																			  );
			END_IF
	ELSE
		 bPumpsMove := TRUE;
	END_IF
	
	IF bPumpsMove THEN
		FOR i := 1 TO 5 DO
			bValvesMove[i] := FALSE;
		END_FOR
		eState := WeightRequest;
	END_IF

// Scale eight request
WeightRequest:
	
	IF NOT bMoveMotorM2 THEN
		bMoveMotorM2 := GVL_Motion.aMotors[2].MoveAbsolute(GVL_Settings.stMachineParam.aM2Position[6], GVL_Settings.stMachineParam.rM2Velocity, GVL_Settings.stMachineParam.rM2Accleration, GVL_Settings.stMachineParam.rM2Deceleration);
	END_IF
	
	IF bMoveMotorM2 THEN
		rScaleWeight := GVL_Calibration.fbScaleDevice.RequestWeight();
	END_IF
	
	IF GVL_Calibration.fbScaleDevice.bWeightReady AND bMoveMotorM2 THEN
		// Fillup Results Array
		GVL_calibration.aDosingResults[iResultRow].iPump	:= iPumpIndex;
		GVL_calibration.aDosingResults[iResultRow].iCheck 	:= iResults;
		GVL_calibration.aDosingResults[iResultRow].rResult 	:= (rScaleWeight - rWeightBefore) / 0.9972;
		GVL_calibration.aDosingResults[iResultRow].iRevs 	:= iRevs;
		rWeightBefore := rScaleWeight;
		rScaleWeight := 0;
		iRevs := 0;
		iResultRow := iResultRow + 1;
		bWeightDone := GVL_Calibration.fbScaleDevice.Reset();
	END_IF
	
	IF bWeightDone THEN
		IF iResults >= iReplicate THEN
			iPumpIndex := iPumpIndex + 1;
			eState := NextPump;
		ELSE
			iResults := iResults + 1;
			eState := MoveValvesSolvent;
		END_IF
	bWeightDone := FALSE;
	bMoveMotorM2 := FALSE;
	END_IF

// Next Pump
NextPump:
	IF iPumpIndex > 10 THEN
		eState := Done;
	ELSE
		IF aPumps[iPumpIndex] THEN
			FOR i := 1 TO 5 DO
				bValvesMove[i] := FALSE;
			END_FOR
			iResults := 1;
			eState := MoveValvesSolvent;
		ELSE
			iPumpIndex := iPumpIndex + 1;
		END_IF	
	END_IF

// Done	
Done:
	bDone := TRUE;
    bBusy := FALSE;
    IF NOT bExecute THEN
        bDone := FALSE;
        eState := Idle;
    END_IF
	
END_CASE

METHOD Reset : BOOL
VAR
	i : USINT;
END_VAR
// Outputs
bDone := FALSE;
bError := FALSE;
bBusy := FALSE;

// Internal control flags
bStartDosing := FALSE;
bWeightDone := FALSE;
bPumpsMove := FALSE;

// Internal indexes / counters
iResults := 1;
iResultRow := 1;
iPumpIndex := 1;

bMoveMotorM2 := FALSE;
bMoveMotorM3 := FALSE;
bExecute := FALSE;

RTrigExecutePulse(CLK := FALSE);

// Internal values
rScaleWeight := 0;

FOR i := 1 TO 5 DO
	bValvesMove[i] := FALSE;
END_FOR

FOR i := 1 TO 10 DO
	rDistanceByVol[i] := 0;
END_FOR

// Return to initial state
eState := Idle;

Reset := TRUE;
END_METHOD

METHOD ResetResults : BOOL
VAR
	i : USINT;
END_VAR
FOR i := 1 TO 100 DO
	GVL_Calibration.aDosingResults[i].iPump 	:= 0;
	GVL_Calibration.aDosingResults[i].iCheck 	:= 0;
	GVL_Calibration.aDosingResults[i].rResult 	:= 0;
	GVL_Calibration.aDosingResults[i].iRevs 	:= 0;
END_FOR

ResetResults := TRUE;
END_METHOD

END_FUNCTION_BLOCK

// ---- POUs/MARCO/DB/DB_Create_Calibration.TcPOU
PROGRAM DB_Create_Calibration
VAR
	state: INT;
	timer: ton;
	i : UDINT;
END_VAR

VAR_INPUT
	start: BOOL;
END_VAR

timer();

CASE state OF
	
0:
	IF start THEN
		DB_Query.state:= E_DB_QUERY_STATE.SELECT_LAST_CALIBRATION_ID;
		timer(in:=TRUE, pt:=T#10S);
		state:= 10;
	ELSE
		state:= 0;
	END_IF

10:

	IF NOT DB_Query.FB_SelectArray.bBusy AND timer.Q THEN
		timer(in:=FALSE);
		GVL_Calibration.stPumpCalibrationInfo.iCalibrationNumber 		:= GVL_DB.lastCalibID[0];	
		GVL_DB.stParameter_PCR.userID									:= 'DEV';
		GVL_DB.stParameter_PCR.allowableFail							:= USINT_TO_STRING(GVL_Settings.stCalibParameters.iAllowableFailures);
		GVL_DB.stParameter_PCR.CalibrationNo							:= UDINT_TO_INT(GVL_Calibration.stPumpCalibrationInfo.iCalibrationNumber+1);
		GVL_DB.stParameter_PCR.callInterval								:= UINT_TO_STRING(GVL_Settings.stCalibParameters.iCalIntervalDays);
		GVL_DB.stParameter_PCR.density									:= REAL_TO_STRING(GVL_Calibration.stPumpCalibrationInfo.rSolventDensity);
		GVL_DB.stParameter_PCR.replicates								:= INT_TO_STRING(GVL_Settings.stCalibParameters.iReplicatesSetpoint);
		GVL_DB.stParameter_PCR.solventNo								:= GVL_Calibration.stPumpCalibrationInfo.iSolventID;
		GVL_DB.stParameter_PCR.solventRevision							:= INT_TO_STRING(GVL_Calibration.stPumpCalibrationInfo.iSolventRevision);
		GVL_DB.stParameter_PCR.sysRevisionNo							:= GVL_Settings.sysRevNumber;	
		state:= 20;
	ELSE
		state:= 10;
	END_IF
	
	// FIX: stamp any measurement that has data but an empty dDateTime.
	// This prevents NULL dates in the database when FB_LocalSystemTime has not
	// yet executed a valid cycle at the moment the measurement was recorded.
	FOR i := 1 TO 100 BY 1 DO
		IF GVL_Calibration.stPumpCalibrationData[i].iPumpNumber > 0 AND
		   GVL_Calibration.stPumpCalibrationData[i].dDateTime = '' THEN
			GVL_Calibration.stPumpCalibrationData[i].dDateTime := GVL_HMI.sDateAndTimeEventTriggered;
		END_IF
	END_FOR
	
20:

	IF TRUE THEN
		DB_Query.state:= E_DB_QUERY_STATE.INSERT_CALIBRATION;
		timer(in:=TRUE, pt:=T#10S);
		state:= 30;
	ELSE
		state:= 20;
	END_IF	

30:

	IF NOT DB_Query.FB_Insert.bBusy AND timer.Q THEN
		timer(in:=FALSE);
		start:= FALSE;
		state:= 0;
	ELSE
		state:= 30;
	END_IF
END_CASE

END_PROGRAM

// ---- POUs/1. MachineControl/PRG_ManualControl.TcPOU
PROGRAM PRG_ManualControl
VAR
	
	rMotorsActualPosition : ARRAY[1..3] OF LREAL;
	rValvesActualPosition : ARRAY[1..5] OF LREAL;
	rPumpsActualPosition  : ARRAY[1..10] OF LREAL;
	rDegreesPerVolume 	  : ARRAY[1..10] OF LREAL;
	
	aPumpsActivated		  : ARRAY[1..10] OF BOOL;
	aPumpsDirection		  : ARRAY[1..10] OF E_PumpDirection;
	aPumpsSpeed			  : ARRAY[1..10] OF REAL;
	aPumpsVolume		  : ARRAY[1..10] OF REAL;
	aPumpsDistance		  : ARRAY[1..10] OF UINT;
	bRunPumpsBySpeed	  : BOOL := FALSE;
	bRunPumpsByVolume	  : BOOL := FALSE;
	bRunPumpsByDistance	  : BOOL := FALSE;
	iM3Position			  : LREAL;
	aMotorBusy	: ARRAY[1..3] OF BOOL;
	
	fbPumpsController : FB_AllPumpsController;

	i : INT; 
	
	//interlock Variables
	iTargetPosM2 : INT;
    rActualPosM3 : LREAL;
    rTol         : LREAL := 3.0; // tolerância para considerar posição "alinhada"
    bAllowMoveM2 : BOOL := TRUE;
		
END_VAR

//Motors Manual jog handling 
MotorsJog();
MotorsActualPosition();

//New Manual Screen commands area ##########################################################
(* <Motors> -----------------------------------------------------------------------------------------------------------------------------------------------------------------------------------*)

(*<M1 Motor>*)
//Move M1 by HMI combobox manual mode
IF GVL_HMI.aManualMotorsCmd[1].bRun THEN
	GVL_HMI.aManualMotorsCmd[1].bRun := NOT GVL_Motion.aMotors[1].MoveAbsolute(	rPosition := GVL_Settings.stMachineParam.aM1Position[GVL_HMI.aManualMotorsCmd[1].iPosition],
                        														rVelocity := GVL_Settings.stMachineParam.rM1Velocity,
                        														rAcc := GVL_Settings.stMachineParam.rM1Accleration,
                       															rDec := GVL_Settings.stMachineParam.rM1Deceleration
																				);
END_IF
//Stop Moviment M1 by HMI manual mode button
IF GVL_HMI.aManualMotorsCmd[1].bStop THEN
	GVL_HMI.aManualMotorsCmd[1].bStop := NOT GVL_Motion.aMotors[1].Stop();
END_IF
(*<\M1 Motor>*)

(*<M2 Motor>*)
//Move M2 by HMI combobox manual mode
iTargetPosM2 := GVL_HMI.aManualMotorsCmd[2].iPosition;
rActualPosM3 := rMotorsActualPosition[3];

//Interlock move for M2 base on M3 position
CASE iTargetPosM2 OF
    3: // Fill Vials
        bAllowMoveM2 := (
            ABS(rActualPosM3 - GVL_Settings.stMachineParam.aM3Position[2]) <= rTol OR //AboveVilSet1
            ABS(rActualPosM3 - (GVL_Settings.stMachineParam.aM3Position[2]+GVL_Settings.stMachineParam.aM3Position[3])) <= rTol OR 	//AboveVilSet2
            ABS(rActualPosM3 - (GVL_Settings.stMachineParam.aM3Position[2]+(2*GVL_Settings.stMachineParam.aM3Position[3]))) <= rTol OR	//AboveVilSet3
            ABS(rActualPosM3 - (GVL_Settings.stMachineParam.aM3Position[2]+(3*GVL_Settings.stMachineParam.aM3Position[3]))) <= rTol		//AboveVilSet4
        );

    4: // Calibration
        bAllowMoveM2 := ABS(rActualPosM3 - GVL_Settings.stMachineParam.aM3Position[4]) <= rTol;

    ELSE
        bAllowMoveM2 := TRUE;
END_CASE

//M2 Moviment if there is no interlock
IF GVL_HMI.aManualMotorsCmd[2].bRun THEN
    IF bAllowMoveM2 THEN
        GVL_HMI.aManualMotorsCmd[2].bRun := NOT GVL_Motion.aMotors[2].MoveAbsolute(
            rPosition := GVL_Settings.stMachineParam.aM2Position[iTargetPosM2],
            rVelocity := GVL_Settings.stMachineParam.rM2Velocity,
            rAcc := GVL_Settings.stMachineParam.rM2Accleration,
            rDec := GVL_Settings.stMachineParam.rM2Deceleration
        );
    ELSE
        GVL_HMI.aManualMotorsCmd[2].bRun := FALSE;
        // TODO: Block flag or alarm
    END_IF
END_IF

//Stop Moviment M2 by HMI manual mode button
IF GVL_HMI.aManualMotorsCmd[2].bStop THEN
	GVL_HMI.aManualMotorsCmd[2].bStop := NOT GVL_Motion.aMotors[2].Stop();
END_IF
(*<\M2 Motor>*)

(*<M3 Motor>*)
//Interlock by M2 Position
IF GVL_HMI.aManualMotorsCmd[3].bRun THEN
    IF ABS(rMotorsActualPosition[2] - GVL_Settings.stMachineParam.aM2Position[1]) > rTol THEN
        //If M2 it is not in Home Position, M3 move cannot be done
        GVL_HMI.aManualMotorsCmd[3].bRun := FALSE;
        // TODO: Block flag or alarm
    ELSE
		CASE GVL_HMI.aManualMotorsCmd[3].iPosition OF 
			1: iM3Position := GVL_Settings.stMachineParam.aM3Position[1];
			2: iM3Position := GVL_Settings.stMachineParam.aM3Position[2];
			3: iM3Position := GVL_Settings.stMachineParam.aM3Position[2] + GVL_Settings.stMachineParam.aM3Position[3];
			4: iM3Position := GVL_Settings.stMachineParam.aM3Position[2] + (2*GVL_Settings.stMachineParam.aM3Position[3]);
			5: iM3Position := GVL_Settings.stMachineParam.aM3Position[2] + (3*GVL_Settings.stMachineParam.aM3Position[3]);
			6: iM3Position := GVL_Settings.stMachineParam.aM3Position[4];
		END_CASE
        GVL_HMI.aManualMotorsCmd[3].bRun := NOT GVL_Motion.aMotors[3].MoveAbsolute(
            rPosition := iM3Position,
            rVelocity := GVL_Settings.stMachineParam.rM3Velocity,
            rAcc := GVL_Settings.stMachineParam.rM3Accleration,
            rDec := GVL_Settings.stMachineParam.rM3Deceleration
        );
    END_IF
END_IF
//Stop Moviment M2 by HMI manual mode button
IF GVL_HMI.aManualMotorsCmd[3].bStop THEN
	GVL_HMI.aManualMotorsCmd[3].bStop := NOT GVL_Motion.aMotors[3].Stop();
END_IF
(*<\M3 Motor>*)

(* <Valves> -----------------------------------------------------------------------------------------------------------------------------------------------------------------------------------*)

(*<Valve 1>*)
//Move Valve 1 by HMI combobox manual mode
IF GVL_HMI.aManualValvesCmd[1].bMove THEN
	GVL_HMI.aManualValvesCmd[1].bMove := NOT GVL_Motion.aValvesObj[1].MoveValve( 	iPosition := GVL_HMI.aManualValvesCmd[1].iTargetPos,
																					rVelocity := GVL_Motion.aValves[1].rTargetVel, 
																					rAcc := GVL_Motion.aValves[1].rAcceleration, 
																					rDec := GVL_Motion.aValves[1].rDeceleration);
END_IF

//Stop Moviment Valve 1 by HMI manual mode button
IF GVL_HMI.aManualValvesCmd[1].bStop THEN
	GVL_HMI.aManualValvesCmd[1].bStop := NOT GVL_Motion.aValvesObj[1].Stop();
END_IF
(*<\Valve 1>*)

(*<Valve 2>*)
//Move Valve 2 by HMI combobox manual mode
IF GVL_HMI.aManualValvesCmd[2].bMove THEN
	GVL_HMI.aManualValvesCmd[2].bMove := NOT GVL_Motion.aValvesObj[2].MoveValve( 	iPosition := GVL_HMI.aManualValvesCmd[2].iTargetPos, 
																					rVelocity := GVL_Motion.aValves[2].rTargetVel, 
																					rAcc := GVL_Motion.aValves[2].rAcceleration, 
																					rDec := GVL_Motion.aValves[2].rDeceleration);
END_IF

//Stop Moviment Valve 2 by HMI manual mode button
IF GVL_HMI.aManualValvesCmd[2].bStop THEN
	GVL_HMI.aManualValvesCmd[2].bStop := NOT GVL_Motion.aValvesObj[2].Stop();
END_IF
(*<\Valve 2>*)

(*<Valve 3>*)
//Move Valve 3 by HMI combobox manual mode
IF GVL_HMI.aManualValvesCmd[3].bMove THEN
	GVL_HMI.aManualValvesCmd[3].bMove := NOT GVL_Motion.aValvesObj[3].MoveValve( 	iPosition := GVL_HMI.aManualValvesCmd[3].iTargetPos, 
																					rVelocity := GVL_Motion.aValves[3].rTargetVel, 
																					rAcc := GVL_Motion.aValves[3].rAcceleration, 
																					rDec := GVL_Motion.aValves[3].rDeceleration);
END_IF

//Stop Moviment Valve 3 by HMI manual mode button
IF GVL_HMI.aManualValvesCmd[3].bStop THEN
	GVL_HMI.aManualValvesCmd[3].bStop := NOT GVL_Motion.aValvesObj[3].Stop();
END_IF
(*<\Valve 3>*)

(*<Valve 4>*)
//Move Valve 4 by HMI combobox manual mode
IF GVL_HMI.aManualValvesCmd[4].bMove THEN
	GVL_HMI.aManualValvesCmd[4].bMove := NOT GVL_Motion.aValvesObj[4].MoveValve( 	iPosition := GVL_HMI.aManualValvesCmd[4].iTargetPos, 
																					rVelocity := GVL_Motion.aValves[4].rTargetVel, 
																					rAcc := GVL_Motion.aValves[4].rAcceleration, 
																					rDec := GVL_Motion.aValves[4].rDeceleration);
END_IF

//Stop Moviment Valve 4 by HMI manual mode button
IF GVL_HMI.aManualValvesCmd[4].bStop THEN
	GVL_HMI.aManualValvesCmd[4].bStop := NOT GVL_Motion.aValvesObj[4].Stop();
END_IF
(*<\Valve 4>*)

(*<Valve 5>*)
//Move Valve 5 by HMI combobox manual mode
IF GVL_HMI.aManualValvesCmd[5].bMove THEN
	GVL_HMI.aManualValvesCmd[5].bMove := NOT GVL_Motion.aValvesObj[5].MoveValve( 	iPosition := GVL_HMI.aManualValvesCmd[5].iTargetPos, 
																					rVelocity := GVL_Motion.aValves[5].rTargetVel, 
																					rAcc := GVL_Motion.aValves[5].rAcceleration, 
																					rDec := GVL_Motion.aValves[5].rDeceleration);
END_IF

//Stop Moviment Valve 5 by HMI manual mode button
IF GVL_HMI.aManualValvesCmd[5].bStop THEN
	GVL_HMI.aManualValvesCmd[5].bStop := NOT GVL_Motion.aValvesObj[5].Stop();
END_IF
(*<\Valve 5>*)

(* <Pumps> -----------------------------------------------------------------------------------------------------------------------------------------------------------------------------------*)
(*<Move by Speed>*)
IF GVL_HMI.bRunPumpsBySpeedBt THEN //Fill up the pump arrays and trigger pumps 
	FOR i := 1 TO 10 DO
		aPumpsActivated[i] := GVL_HMI.aManualPumpsCmd[i].bActive;
		aPumpsDirection[i] := GVL_HMI.aManualPumpsCmd[i].eDirection;
		aPumpsSpeed[i] := GVL_HMI.aManualPumpsCmd[i].rSpeed * 6;
	END_FOR
	bRunPumpsBySpeed := TRUE;
	GVL_HMI.bRunPumpsBySpeedBt := FALSE;
END_IF
IF bRunPumpsBySpeed THEN //pumps movement
	bRunPumpsBySpeed := NOT fbPumpsController.MoveBySpeed(aPumpIds := aPumpsActivated, aVelocity := aPumpsSpeed, aPumpDirection := aPumpsDirection);
END_IF
(*<\Move by Speed>*)

(*<Move by Volume>*)
IF GVL_HMI.bRunPumpsByVolumeBt THEN //Fill up the pump arrays and trigger pumps 
	FOR i := 1 TO 10 DO
		aPumpsActivated[i] := GVL_HMI.aManualPumpsCmd[i].bActive;
		aPumpsDirection[i] := GVL_HMI.aManualPumpsCmd[i].eDirection;
		aPumpsSpeed[i] := GVL_HMI.aManualPumpsCmd[i].rSpeed * 6;
		aPumpsVolume[i] := GVL_HMI.aManualPumpsCmd[i].rVolume;
	END_FOR
	bRunPumpsByVolume := TRUE;
	GVL_HMI.bRunPumpsByVolumeBt := FALSE;
END_IF
IF bRunPumpsByVolume THEN //pumps movement
	bRunPumpsByVolume := NOT fbPumpsController.MoveByVolume(aPumpIds := aPumpsActivated, aVolume := aPumpsVolume, aPumpDirection := aPumpsDirection, aVelocity := aPumpsSpeed);
END_IF
(*<\Move by Volume>*)

(*<Move by Distance>*)
IF GVL_HMI.bRunPumpsByDistanceBt THEN //Fill up the pump arrays and trigger pumps 
	FOR i := 1 TO 10 DO
		aPumpsActivated[i] := GVL_HMI.aManualPumpsCmd[i].bActive;
		aPumpsDirection[i] := GVL_HMI.aManualPumpsCmd[i].eDirection;
		aPumpsSpeed[i] := GVL_HMI.aManualPumpsCmd[i].rSpeed * 6;
		aPumpsDistance[i] := GVL_HMI.aManualPumpsCmd[i].iDistance;
	END_FOR
	bRunPumpsByDistance := TRUE;
	GVL_HMI.bRunPumpsByDistanceBt := FALSE;
END_IF
IF bRunPumpsByDistance THEN //pumps movement
	bRunPumpsByDistance := NOT fbPumpsController.MoveByDistance(aPumpIds := aPumpsActivated, aRevolutions := aPumpsDistance, aPumpDirection := aPumpsDirection, aVelocity := aPumpsSpeed);
END_IF
(*<\Move by Distance>*)

(*<Stop All Pumps>*)
IF GVL_HMI.bStopPumpsBt THEN
	GVL_HMI.bStopPumpsBt := NOT fbPumpsController.StopAllPumps();
END_IF
(*<\Stop All Pumps>*)

(* <\Pumps> ----------------------------------------------------------------------------------------------------------------------------------------------------------------------------------*)

